(* CODESYS project SMART_HOME_SANDBOX_V2.xml

Project tree, tasks and I/O mapping:
  PLC_A : PLC210, Production association OWEN, order no. 1, version 3.5.17.35
    application Application
      libraries: SysMem, 3.5.17.0 (System); Net Base Services, 3.5.17.0 (3S - Smart Software Solutions GmbH); OwenCommunication, 3.5.11.7 (Production association OWEN); Standard, * (System); AC_ModuleBase, * (3S - Smart Software Solutions GmbH); AC_DataLog, * (3S - Smart Software Solutions GmbH); VisuElem3DPath, 4.1.0.0 (System); VisuElemMeter, 4.1.0.0 (System); VisuElemTrace, 4.1.0.0 (System); VisuElemBase, 4.1.0.0 (System); VisuElems, 4.1.0.0 (System); VisuElemsSpecialControls, 4.1.0.0 (System); VisuElemsWinControls, 4.1.0.0 (System); VisuElemTextEditor, 4.1.0.0 (System); VisuNativeControl, 4.1.0.0 (System); VisuElemsAlarm, 4.1.0.0 (System); VisuElemCamDisplayer, 4.1.0.0 (System); VisuElemsDateTime, 4.1.0.0 (System); VisuElemXYChart, 4.1.0.0 (System); VisuInputs, 4.1.0.0 (System); CmpTargetVisu, 3.5.17.0 (System); Mx210 Assistant, 3.5.11.11 (Production association OWEN)
      task MainTask (cyclic, interval t#20ms, priority 1) calls PRG_PLC_A, PRG_PLC_B, PRG_Main
      task OwenCloudTask (cyclic, interval T#25ms, priority 31) calls OwenStorage.CLOUD_PRG
      task VISU_TASK (cyclic, interval 100 ms, priority 31) calls VisuElems.Visu_Prg
      program PRG_PLC_A [ST]
      program PRG_PLC_B [ST]
    Ethernet : Ethernet, 3S - Smart Software Solutions GmbH, version 3.5.17.0
        settings: IPAddress = [192,168,10,10]; SubnetMask = [255,255,255,0]; GatewayAddress = [192,168,10,1]; MACAddress = [16#00,16#00,16#00,16#00,16#00,16#00]; NetworkInterfaceName = 'ELECTRICAL_ROOM_1F'; NetworkInterfaceName = "ELECTRICAL_ROOM_1F"; SaveCommunicationSettings = TRUE
      Modbus_TCP_Master : Modbus TCP Master, 3S - Smart Software Solutions GmbH, version 3.5.17.0
        MV210_101 : MV210-101, Production association OWEN, version 3.5.11.13
            settings: Unit-ID = 2; IPAddress = [192, 168, 10, 2]
            input  Application.GVL_IO.AI_Temp_Outdoor : InputValue  // Вход 1
            input  Application.GVL_IO.AI_Temp_Outdoor : REAL  // Вход 1.Значение
            input  Application.GVL_IO.AI_Manifold_Temps_Supply[1] : InputValue  // Вход 2
            input  Application.GVL_IO.AI_Manifold_Temps_Supply[1] : REAL  // Вход 2.Значение
            input  Application.GVL_IO.AI_Manifold_Temps_Supply[2] : InputValue  // Вход 3
            input  Application.GVL_IO.AI_Manifold_Temps_Supply[2] : REAL  // Вход 3.Значение
            input  Application.GVL_IO.AI_Manifold_Temps_Supply[3] : InputValue  // Вход 4
            input  Application.GVL_IO.AI_Manifold_Temps_Supply[3] : REAL  // Вход 4.Значение
            input  Application.GVL_IO.AI_Manifold_Temps_Supply[4] : InputValue  // Вход 5
            input  Application.GVL_IO.AI_Manifold_Temps_Supply[4] : REAL  // Вход 5.Значение
            input  Application.GVL_IO.AI_Manifold_Temps_Supply[5] : InputValue  // Вход 6
            input  Application.GVL_IO.AI_Manifold_Temps_Supply[5] : REAL  // Вход 6.Значение
            input  Application.GVL_IO.AI_Methane_LEL[1] : InputValue  // Вход 7
            input  Application.GVL_IO.AI_Methane_LEL[1] : REAL  // Вход 7.Значение
            input  Application.GVL_IO.AI_Methane_LEL[2] : InputValue  // Вход 8
            input  Application.GVL_IO.AI_Methane_LEL[2] : REAL  // Вход 8.Значение
            unmapped channels: Tmp, Исключить модуль из опроса, Флаг ошибки, Записать настройки, Прочитать настройки, Вход 1 (чтение), Вход 2 (чтение), Вход 3 (чтение), Вход 4 (чтение), Вход 5 (чтение), Вход 6 (чтение), Вход 7 (чтение), Вход 8 (чтение), Вход 1 (запись), Вход 2 (запись), Вход 3 (запись), Вход 4 (запись), Вход 5 (запись), Вход 6 (запись), Вход 7 (запись), Вход 8 (запись)
        MK210_301 : MK210-301, Production association OWEN, version 3.5.11.13
            settings: Unit-ID = 3; IPAddress = [192, 168, 10, 3]
            input  Application.GVL_IO.DI_Security_Open[1] : BOOL  // Битовая маска входов.Вход 1
            input  Application.GVL_IO.DI_Security_Open[2] : BOOL  // Битовая маска входов.Вход 2
            input  Application.GVL_IO.DI_Security_Open[3] : BOOL  // Битовая маска входов.Вход 3
            input  Application.GVL_IO.DI_Security_Open[4] : BOOL  // Битовая маска входов.Вход 4
            input  Application.GVL_IO.DI_Security_Open[5] : BOOL  // Битовая маска входов.Вход 5
            input  Application.GVL_IO.DI_Security_Open[6] : BOOL  // Битовая маска входов.Вход 6
            input  Application.GVL_IO.DO_Manifold_Pumps[1] : BOOL  // Битовая маска выходов (чтение).Выход 1
            input  Application.GVL_IO.DO_Manifold_Pumps[2] : BOOL  // Битовая маска выходов (чтение).Выход 2
            input  Application.GVL_IO.DO_Manifold_Pumps[3] : BOOL  // Битовая маска выходов (чтение).Выход 3
            input  Application.GVL_IO.DO_Manifold_Pumps[4] : BOOL  // Битовая маска выходов (чтение).Выход 4
            input  Application.GVL_IO.DO_Manifold_Pumps[5] : BOOL  // Битовая маска выходов (чтение).Выход 5
            input  Application.GVL_IO.DO_Boiler_Enable[1] : BOOL  // Битовая маска выходов (чтение).Выход 6
            input  Application.GVL_IO.DO_Boiler_Enable[2] : BOOL  // Битовая маска выходов (чтение).Выход 7
            output Application.GVL_IO.DO_Manifold_Pumps[1] : BOOL  // Битовая маска выходов (запись).Выход 1
            output Application.GVL_IO.DO_Manifold_Pumps[2] : BOOL  // Битовая маска выходов (запись).Выход 2
            output Application.GVL_IO.DO_Manifold_Pumps[3] : BOOL  // Битовая маска выходов (запись).Выход 3
            output Application.GVL_IO.DO_Manifold_Pumps[4] : BOOL  // Битовая маска выходов (запись).Выход 4
            output Application.GVL_IO.DO_Manifold_Pumps[5] : BOOL  // Битовая маска выходов (запись).Выход 5
            output Application.GVL_IO.DO_Boiler_Enable[1] : BOOL  // Битовая маска выходов (запись).Выход 6
            output Application.GVL_IO.DO_Boiler_Enable[2] : BOOL  // Битовая маска выходов (запись).Выход 7
            output Application.GVL_IO.DO_DHW_Heating_Pump : BOOL  // Битовая маска выходов (запись).Выход 8
            output Application.GVL_IO.AO_Supply_Fans[1] : localTypes:PwmOutputValue  // Коэффициент заполнения ШИМ (запись)
            output Application.GVL_IO.AO_Supply_Fans[2] : localTypes:PwmOutputValue  // Коэффициент заполнения ШИМ (запись)
            output Application.GVL_IO.AO_Supply_Fans[3] : localTypes:PwmOutputValue  // Коэффициент заполнения ШИМ (запись)
            output Application.GVL_IO.AO_Exhaust_Fans[1] : localTypes:PwmOutputValue  // Коэффициент заполнения ШИМ (запись)
            output Application.GVL_IO.AO_Exhaust_Fans[2] : localTypes:PwmOutputValue  // Коэффициент заполнения ШИМ (запись)
            output Application.GVL_IO.AO_Exhaust_Fans[3] : localTypes:PwmOutputValue  // Коэффициент заполнения ШИМ (запись)
            output Application.GVL_IO.AO_Exhaust_Fans[4] : localTypes:PwmOutputValue  // Коэффициент заполнения ШИМ (запись)
            output Application.GVL_IO.AO_Exhaust_Fans[5] : localTypes:PwmOutputValue  // Коэффициент заполнения ШИМ (запись)
            unmapped channels: Tmp, Исключить модуль из опроса, Флаг ошибки, Битовая маска входов, Битовая маска выходов (чтение), Битовая маска выходов (запись), Значение счетчика, Значение счетчика, Значение счетчика, Значение счетчика, Значение счетчика, Значение счетчика, Сбросить счетчик, Сбросить счетчик, Сбросить счетчик, Сбросить счетчик, Сбросить счетчик, Сбросить счетчик, Период ШИМ (чтение), Период ШИМ (чтение), Период ШИМ (чтение), Период ШИМ (чтение), Период ШИМ (чтение), Период ШИМ (чтение), Период ШИМ (чтение), Период ШИМ (чтение), Период ШИМ (запись), Период ШИМ (запись), Период ШИМ (запись), Период ШИМ (запись), Период ШИМ (запись), Период ШИМ (запись), Период ШИМ (запись), Период ШИМ (запись), Коэффициент заполнения ШИМ (чтение), Коэффициент заполнения ШИМ (чтение), Коэффициент заполнения ШИМ (чтение), Коэффициент заполнения ШИМ (чтение), Коэффициент заполнения ШИМ (чтение), Коэффициент заполнения ШИМ (чтение),
              Коэффициент заполнения ШИМ (чтение), Коэффициент заполнения ШИМ (чтение)
        MV210_202 : MV210-202, Production association OWEN, version 3.5.11.13
            settings: Unit-ID = 4; IPAddress = [192, 168, 10, 4]
            input  Application.GVL_IO.DI_Flood_Sensors[1] : BOOL  // Битовая маска входов.Вход 1
            input  Application.GVL_IO.DI_Flood_Sensors[2] : BOOL  // Битовая маска входов.Вход 2
            input  Application.GVL_IO.DI_Flood_Sensors[3] : BOOL  // Битовая маска входов.Вход 3
            input  Application.GVL_IO.DI_Flood_Sensors[4] : BOOL  // Битовая маска входов.Вход 4
            input  Application.GVL_IO.DI_Flood_Sensors[5] : BOOL  // Битовая маска входов.Вход 5
            input  Application.GVL_IO.DI_Flood_Sensors[6] : BOOL  // Битовая маска входов.Вход 6
            input  Application.GVL_IO.DI_Flood_Sensors[7] : BOOL  // Битовая маска входов.Вход 7
            input  Application.GVL_IO.DI_Flood_Sensors[8] : BOOL  // Битовая маска входов.Вход 8
            input  Application.GVL_IO.DI_Flood_Sensors[9] : BOOL  // Битовая маска входов.Вход 9
            input  Application.GVL_IO.DI_Flood_Sensors[10] : BOOL  // Битовая маска входов.Вход 10
            input  Application.GVL_IO.DI_Flood_Sensors[11] : BOOL  // Битовая маска входов.Вход 11
            input  Application.GVL_IO.DI_Flood_Sensors[12] : BOOL  // Битовая маска входов.Вход 12
            input  Application.GVL_IO.DI_Security_Glass[1] : BOOL  // Битовая маска входов.Вход 13
            input  Application.GVL_IO.DI_Security_Glass[2] : BOOL  // Битовая маска входов.Вход 14
            input  Application.GVL_IO.DI_Security_Glass[3] : BOOL  // Битовая маска входов.Вход 15
            input  Application.GVL_IO.DI_Security_Glass[4] : BOOL  // Битовая маска входов.Вход 16
            input  Application.GVL_IO.DI_Security_Glass[5] : BOOL  // Битовая маска входов.Вход 17
            input  Application.GVL_IO.DI_Security_Glass[6] : BOOL  // Битовая маска входов.Вход 18
            input  Application.GVL_IO.DI_Security_Glass[7] : BOOL  // Битовая маска входов.Вход 19
            input  Application.GVL_IO.DI_Security_Glass[8] : BOOL  // Битовая маска входов.Вход 20
            unmapped channels: Tmp, Исключить модуль из опроса, Флаг ошибки, Битовая маска входов, Значение, Значение, Значение, Значение, Значение, Значение, Значение, Значение, Значение счетчика, Значение счетчика, Значение счетчика, Значение счетчика, Значение счетчика, Значение счетчика, Значение счетчика, Значение счетчика, Значение счетчика, Значение счетчика, Значение счетчика, Значение счетчика, Сбросить значение, Сбросить значение, Сбросить значение, Сбросить значение, Сбросить значение, Сбросить значение, Сбросить значение, Сбросить значение, Сбросить счетчик, Сбросить счетчик, Сбросить счетчик, Сбросить счетчик, Сбросить счетчик, Сбросить счетчик, Сбросить счетчик, Сбросить счетчик,
              Сбросить счетчик, Сбросить счетчик, Сбросить счетчик, Сбросить счетчик
        MU210_401 : MU210-401, Production association OWEN, version 3.5.11.13
            settings: Unit-ID = 5; IPAddress = [192, 168, 10, 5]
            output Application.GVL_IO.AO_Manifold_Valves[1] : localTypes:CoefficientPWM  // Коэффициент заполнения ШИМ (запись)
            output Application.GVL_IO.AO_Manifold_Valves[2] : localTypes:CoefficientPWM  // Коэффициент заполнения ШИМ (запись)
            output Application.GVL_IO.AO_Manifold_Valves[3] : localTypes:CoefficientPWM  // Коэффициент заполнения ШИМ (запись)
            output Application.GVL_IO.AO_Manifold_Valves[4] : localTypes:CoefficientPWM  // Коэффициент заполнения ШИМ (запись)
            output Application.GVL_IO.AO_Manifold_Valves[5] : localTypes:CoefficientPWM  // Коэффициент заполнения ШИМ (запись)
            output Application.GVL_IO.AO_Boiler_Setpoint[1] : localTypes:CoefficientPWM  // Коэффициент заполнения ШИМ (запись)
            output Application.GVL_IO.AO_Boiler_Setpoint[2] : localTypes:CoefficientPWM  // Коэффициент заполнения ШИМ (запись)
            unmapped channels: Tmp, Исключить модуль из опроса, Флаг ошибки, Битовая маска выходов (чтение), Битовая маска выходов (запись), Период ШИМ (чтение), Период ШИМ (чтение), Период ШИМ (чтение), Период ШИМ (чтение), Период ШИМ (чтение), Период ШИМ (чтение), Период ШИМ (чтение), Период ШИМ (чтение), Период ШИМ (запись), Период ШИМ (запись), Период ШИМ (запись), Период ШИМ (запись), Период ШИМ (запись), Период ШИМ (запись), Период ШИМ (запись), Период ШИМ (запись), Коэффициент заполнения ШИМ (чтение), Коэффициент заполнения ШИМ (чтение), Коэффициент заполнения ШИМ (чтение), Коэффициент заполнения ШИМ (чтение), Коэффициент заполнения ШИМ (чтение), Коэффициент заполнения ШИМ (чтение), Коэффициент заполнения ШИМ (чтение), Коэффициент заполнения ШИМ (чтение), Коэффициент заполнения ШИМ (запись)
    PLC210_11 : PLC210-11, Production association OWEN, version 3.5.17.3004
        unmapped channels: Канал питания 1, Канал питания 2, Сервисная кнопка, Температура CPU, Переключатель Старт\Стоп, Напряжение батареи часов, Статус батареи часов, Статус ионисторов, Hostname, New Hostame, Set Hostname
      LeftSide : LeftSide-11, Production association OWEN, version 3.5.17.3004
          unmapped channels: Битовая маска входов, Cчётчик импульсов, Cчётчик импульсов, Cчётчик импульсов, Cчётчик импульсов, Cчётчик импульсов, Cчётчик импульсов, Cчётчик импульсов, Cчётчик импульсов, Период импульса, Период импульса, Период импульса, Период импульса, Период импульса, Период импульса, Период импульса, Период импульса, Длительность импульса, Длительность импульса, Длительность импульса, Длительность импульса, Длительность импульса, Длительность импульса, Длительность импульса, Длительность импульса, Статус генератора импульсов, Статус генератора импульсов, Статус генератора импульсов, Статус генератора импульсов, Осталось сгенерировать импульсов, Осталось сгенерировать импульсов, Осталось сгенерировать импульсов, Осталось сгенерировать импульсов, Сброс счётчика импульсов, Сброс счётчика импульсов, Сброс счётчика импульсов, Сброс счётчика импульсов, Сброс счётчика импульсов, Сброс счётчика импульсов, Сброс счётчика импульсов,
            Сброс счётчика импульсов, Битовая маска выходов (запись), Запустить генератор, Запустить генератор, Запустить генератор, Запустить генератор, Количество импульсов генератора (запись), Количество импульсов генератора (запись), Количество импульсов генератора (запись), Количество импульсов генератора (запись), Выход 1, Выход 2, Выход 3, Выход 4, Выход 1, Выход 2, Выход 3, Выход 4, Выход 1, Выход 2, Выход 3, Выход 4, Выход 1, Выход 2, Выход 3, Выход 4
      RightSide : RightSide-11, Production association OWEN, version 3.5.17.3002
          unmapped channels: Наличие связи, Счетчик ошибок, Битовая маска диагностики выходов, Битовая маска выходов (запись)
    OwenRTC : OwenRTC, Production association OWEN, version 3.5.17.3002
        unmapped channels: Year, Month, Day, Hour, Minute, Second, Day of Week, Week of Year, Format Date, Format Time, UTC Offset, NTP Enabled, NTP Error, System Timer, Date And Time, Operating Time, New Year, New Month, New Day, New Hour, New Minute, New Second, New UTC Offset, Set Settings DT, Enable NTP, Prefer Server, Sync time by NTP
    OwenCloud : OwenCloud, Production association OWEN, version 3.5.17.3004
        unmapped channels: OwenCloud enabled, Folder error, Symbol error, No Symbol Config, Status, Warning Big Symbol Name, Warning Symbol Name, Symbol Count, Enable OwenCloud
    Buzzer : Buzzer, Production association OWEN, version 3.5.17.3002
        unmapped channels: Buzzer enabled, Enable Buzzer, Sound frequency
    Drives : Drives, Production association OWEN, version 3.5.17.3003
        unmapped channels: FS size, FS used, FS free, USB Mounted, USB Unmount done, USB size, USB used, USB free, MMC Mounted, MMC Unmount done, MMC size, MMC used, MMC free, FS wear, USB FS Info, MMC FS Info, Enable Drives, USB Unmount, MMC Unmount
    Debug : Debug, Production association OWEN, version 3.5.17.3002
        unmapped channels: RAM used, RAM free, Open files, Processor usage, Core temp, Enable Debug, Debug pause
    Info : Info, Production association OWEN, version 3.5.17.3002
        unmapped channels: VENDOR, DEVICE, SERIAL, RUNTIME, FIRMWARE, LINUX, TARGET, PROJECT, AUTHOR, VERSION, PROFILE, LASTCHANGES
    Watchdog : Watchdog, Production association OWEN, version 3.5.17.3002
        unmapped channels: Exception Handling, Last Exception Code, Last Exception Description, Last Exception Time, Hardware Watchdog Flag, Power Reboot Count, Watchdog Reboot Count, Exception Reboot Count, Command Reboot Count, Reboot, Reset Counters
  libraries: VisuSymbols, 4.1.0.0 (System); SysFileAsync, 3.5.17.0 (System); SysFile, 3.5.17.0 (System); Mx210 Assistant, 3.5.11.11 (Production association OWEN); VisuElemsDateTime Interfaces, 4.1.0.0 (Intern)
  DUT/
    ENUM/
      data type E_ALERT_PRIORITY
      data type E_Debug_Log_Level
      data type E_Lifetime_Device_Type
      data type E_Outdoor_Mode
      data type E_PLC_ROLE
      data type E_Rule_Action_Type
      data type E_Rule_Comparison
      data type E_Rule_Condition_Type
      data type E_SCENARIO_TYPE
      data type E_SENSOR_TYPE
      data type E_Trend_Parameter_Type
      data type E_TwoFactor_Method
      data type E_Valve_Test_Result
      data type E_VALVE_TYPE
      data type E_VENTILATION_LOCATION
      data type E_VENTILATION_UNIT_TYPE
      data type E_WEATHER_COMPENSATION_METHOD
      data type E_Zone_Access_Level
    STRUCT/
      data type ST_Astro_Time
      data type ST_BlackBox_Record
      data type ST_Boiler_Status
      data type ST_Component_Maintenance
      data type ST_Debug_Logger_Config
      data type ST_Debug_Log_Record
      data type ST_Device_Health
      data type ST_DHW_Config
      data type ST_DHW_Status
      data type ST_Flood_Config
      data type ST_Flood_Global_Config
      data type ST_FloorHeating_Circuit_Config
      data type ST_FloorHeating_Global_Config
      data type ST_FloorHeating_Manifold_Config
      data type ST_Gas_Valve_Configuration
      data type ST_Gateway_Command
      data type ST_Heating_Config
      data type ST_History_Record
      data type ST_Lifetime_Status
      data type ST_Maintenance_Access_Config
      data type ST_Manifold_Status
      data type ST_Operator_Zone_Rights
      data type ST_Outdoor_Zone_Config
      data type ST_Owen_Analog_Value
      data type ST_Rule_Action
      data type ST_Scenario_Config
      data type ST_Scenario_Transition_Config
      data type ST_Security_Config
      data type ST_Security_Global_Config
      data type ST_Security_Zone_State
      data type ST_Sensor_Calibration_Record
      data type ST_State_Snapshot
      data type ST_System_State_Summary
      data type ST_Tariff_Config
      data type ST_Trend_Config
      data type ST_Trend_Data
      data type ST_Trend_Header
      data type ST_Trend_History_Record
      data type ST_TwoFactor_Auth_State
      data type ST_TwoFactor_Data
      data type ST_User_Rule
      data type ST_Valve_Test_Config
      data type ST_Ventilation_Config
      data type ST_Ventilation_Global_Config
      data type ST_Ventilation_Scenario_Mode
      data type ST_Ventilation_Unit
      data type ST_Ventilation_Unit_Config
      data type ST_Zone_Sensors
  GVL/
    global variables GVL_BlackBox
    global variables GVL_Constants
    global variables GVL_Diagnostics
    global variables GVL_Global_Variables
    global variables GVL_HMI_Config
    global variables GVL_IO
    global variables GVL_Vars
  POUs/
    function block FB_AccessCode_Manager [ST]
    function block FB_Access_Control [ST]
    function block FB_Astro_Timer [ST]
    function block FB_BlackBox_Recorder [ST]
    function block FB_Boiler_Cascade_Controller [ST]
    function block FB_Boiler_Cascade_Manager [ST]
    function block FB_Calibration_Manager [ST]
    function block FB_CO_Detector [ST]
    function block FB_CRC32_Calculator [ST]: Calculate, InitTable
    function block FB_Debug_Logger [ST]
    function block FB_Device_Predictive_Diag [ST]
    function block FB_DHW_Manager [ST]
    function block FB_Emergency_Valve_Open [ST]
    function block FB_Exhaust_Ventilation_Controller [ST]
    function block FB_Flood_Detector [ST]
    function block FB_FloorHeating_Controller [ST]
    function block FB_FloorHeating_Freeze_Protection [ST]
    function block FB_FloorHeating_Overheat_Protection [ST]
    function block FB_Gas_Methane_Detector [ST]
    function block FB_Gas_Smoke_Manager [ST]
    function block FB_Gas_Valve_Controller [ST]: CloseValve, GetStatus, OpenValve
    function block FB_Gateway_Interface [ST]
    function block FB_Heating_System_Manager [ST]
    function block FB_History_Manager [ST]
    function block FB_Lifetime_Predictor [ST]
    function block FB_Lighting_Blinds_Manager [ST]
    function block FB_Maintenance_Access [ST]
    function block FB_Manifold_Mixing_Valve_Controller [ST]
    function block FB_Manifold_Pump_Controller [ST]
    function block FB_Manual_Valve_Control [ST]
    function block FB_NVRAM_Manager [ST]
    function block FB_Outdoor_Lighting_Controller [ST]
    function block FB_PID_Controller [ST]
    function block FB_PLC_Heartbeat [ST]
    function block FB_Presence_Playback [ST]
    function block FB_Presence_Simulator [ST]
    function block FB_Pre_Departure_Heating [ST]
    function block FB_Random_Generator [ST]: Random_Int_Range
    function block FB_Scenario_Manager [ST]
    function block FB_Scenario_Transition_Controller [ST]
    function block FB_Security_Alarm [ST]: CheckPerimeter
    function block FB_Security_System [ST]
    function block FB_Security_System_Manager [ST]
    function block FB_Sensor_Calibration_Processor [ST]
    function block FB_Sensor_Distribution [ST]
    function block FB_Simulation_Manager [ST]
    function block FB_Smoke_Detector [ST]
    function block FB_SMS_Notification [ST]
    function block FB_State_Manager [ST]
    function block FB_State_Snapshot_Manager [ST]
    function block FB_State_Snapshot_NVRAM [ST]
    function block FB_Supply_Ventilation_Controller [ST]
    function block FB_Trend_Analyzer [ST]
    function block FB_TwoFactor_Auth [ST]
    function block FB_User_Rule_Engine [ST]
    function block FB_Valve_Test [ST]
    function block FB_Ventilation_System_Manager [ST]
    function block FB_Water_Leakage_Manager [ST]
    function block FB_Water_Valve_Controller [ST]: CloseValve, GetStatus, OpenValve
    function block FB_Zone_Access_Manager [ST]: CheckAccess
  text list GlobalTextList
  interface IValveController: CloseValve, GetStatus, OpenValve
  program PRG_Main [ST]
  visualisation Visualization
*)

// DUT/ENUM/E_ALERT_PRIORITY
{attribute 'qualified_only'}
{attribute 'strict'}
TYPE E_ALERT_PRIORITY :
(
    ALERT_PRIORITY_NONE := 0,
    ALERT_PRIORITY_LOW := 1,
    ALERT_PRIORITY_MEDIUM := 2,
    ALERT_PRIORITY_HIGH := 3,
    ALERT_PRIORITY_CRITICAL := 4
) BYTE;
END_TYPE

// DUT/ENUM/E_Debug_Log_Level
{attribute 'qualified_only'}
{attribute 'strict'}
TYPE E_Debug_Log_Level :
(
    LOG_LEVEL_MINIMAL := 0,
    LOG_LEVEL_NORMAL := 1,
    LOG_LEVEL_VERBOSE := 2,
    LOG_LEVEL_DEBUG := 3
) BYTE;
END_TYPE

// DUT/ENUM/E_Lifetime_Device_Type
{attribute 'qualified_only'}
{attribute 'strict'}
TYPE E_Lifetime_Device_Type :
(
    LIFETIME_DEVICE_PUMP := 1,
    LIFETIME_DEVICE_FAN  := 2
) BYTE;
END_TYPE

// DUT/ENUM/E_Outdoor_Mode
{attribute 'qualified_only'}
{attribute 'strict'}
TYPE E_Outdoor_Mode :
(
    OUTDOOR_MODE_AUTO := 0,
    OUTDOOR_MODE_PARTY := 1,
    OUTDOOR_MODE_SECURITY := 2,
    OUTDOOR_MODE_ECONOMY := 3,
    OUTDOOR_MODE_MANUAL := 4
) BYTE;
END_TYPE

// DUT/ENUM/E_PLC_ROLE
{attribute 'qualified_only'}
{attribute 'strict'}
TYPE E_PLC_ROLE :
(
    ROLE_UNDEFINED := 0,
    ROLE_ACTIVE := 1,
    ROLE_STANDBY := 2,
    ROLE_OFFLINE := 3
) USINT;
END_TYPE

// DUT/ENUM/E_Rule_Action_Type
{attribute 'qualified_only'}
{attribute 'strict'}
TYPE E_Rule_Action_Type :
(
    ACTION_NONE := 0,
    ACTION_SET_FLOOR_HEATING := 1,
    ACTION_SET_LIGHTING_BASE := 2,
    ACTION_SET_LIGHTING_ACCENT := 3,
    ACTION_SET_SOCKET := 4,
    ACTION_SET_VENTILATION := 5,
    ACTION_SET_BLINDS := 6,
    ACTION_ACTIVATE_SCENARIO := 7,
    ACTION_TOGGLE_LIGHTING := 8,
    ACTION_TOGGLE_SOCKET := 9
) BYTE;
END_TYPE

// DUT/ENUM/E_Rule_Comparison
{attribute 'qualified_only'}
{attribute 'strict'}
TYPE E_Rule_Comparison :
(
    COMP_NONE := 0,
    COMP_EQ := 1,
    COMP_GT := 2,
    COMP_LT := 3,
    COMP_GE := 4,
    COMP_LE := 5,
    COMP_IN_RANGE := 6,
    COMP_TRUE := 7,
    COMP_FALSE := 8
) BYTE;
END_TYPE

// DUT/ENUM/E_Rule_Condition_Type
{attribute 'qualified_only'}
{attribute 'strict'}
TYPE E_Rule_Condition_Type :
(
    COND_NONE := 0,
    COND_AIR_TEMP := 1,
    COND_FLOOR_TEMP := 2,
    COND_HUMIDITY := 3,
    COND_CO2 := 4,
    COND_METHANE := 5,
    COND_CO := 6,
    COND_DOOR_WINDOW := 7,
    COND_FLOOD := 8,
    COND_SMOKE := 9,
    COND_MOTION := 10,
    COND_TIME_OF_DAY := 11,
    COND_DAY_OF_WEEK := 12,
    COND_AND := 13, // Логическое И (Rule Chaining)
    COND_OR := 14   // Логическое ИЛИ (Rule Chaining)
) BYTE;
END_TYPE

// DUT/ENUM/E_SCENARIO_TYPE
{attribute 'qualified_only'}
{attribute 'strict'}
TYPE E_SCENARIO_TYPE :
(
    SCENARIO_NONE := 0,
    SCENARIO_MORNING := 1,
    SCENARIO_EVENING := 2,
    SCENARIO_AWAY := 3,
    SCENARIO_PARTY := 4,
    SCENARIO_SLEEP := 5,
    SCENARIO_EMERGENCY := 6,
    SCENARIO_PRESENCE := 7
) BYTE;
END_TYPE

// DUT/ENUM/E_SENSOR_TYPE
{attribute 'qualified_only'}
{attribute 'strict'}
TYPE E_SENSOR_TYPE :
(
  SENSOR_TYPE_NONE := 0,
  SENSOR_TYPE_DOOR_WINDOW := 5,
  SENSOR_TYPE_GLASS_BREAK := 6,
  SENSOR_TYPE_FLOOD := 7,
  SENSOR_TYPE_SMOKE := 8,
  SENSOR_TYPE_GAS_METHANE := 1,
  SENSOR_TYPE_GAS_CO := 2,
  SENSOR_TYPE_TEMP_FLOOR := 3,
  SENSOR_TYPE_TEMP_AIR := 4
) USINT;
END_TYPE

// DUT/ENUM/E_Trend_Parameter_Type
{attribute 'qualified_only'}
{attribute 'strict'}
TYPE E_Trend_Parameter_Type :
(
    TREND_PARAM_NONE := 0,
    TREND_PARAM_TEMP_AIR := 1,
    TREND_PARAM_TEMP_FLOOR := 2,
    TREND_PARAM_PRESSURE := 3,
    TREND_PARAM_PUMP_CURRENT := 4,
    TREND_PARAM_GAS_METHANE := 5,
    TREND_PARAM_GAS_CO := 6
) BYTE;
END_TYPE

// DUT/ENUM/E_TwoFactor_Method
{attribute 'qualified_only'}
{attribute 'strict'}
TYPE E_TwoFactor_Method :
(
    TF_METHOD_NONE := 0,
    TF_METHOD_RFID := 1,
    TF_METHOD_TOTP := 2,
    TF_METHOD_BOTH := 3
) BYTE;
END_TYPE

// DUT/ENUM/E_Valve_Test_Result
{attribute 'qualified_only'}
{attribute 'strict'}
TYPE E_Valve_Test_Result :
(
    TEST_RESULT_NONE := 0,
    TEST_RESULT_PASSED := 1,
    TEST_RESULT_CURRENT_DEVIATION := 2,
    TEST_RESULT_TIME_DEVIATION := 3,
    TEST_RESULT_STALL := 4,
    TEST_RESULT_LIMIT_SWITCH_FAIL := 5,
    TEST_RESULT_ABORTED := 6
) BYTE;
END_TYPE

// DUT/ENUM/E_VALVE_TYPE
{attribute 'qualified_only'}
{attribute 'strict'}
TYPE E_VALVE_TYPE :
(
  VALVE_NC := 1,  // Нормально-закрытый
  VALVE_NO := 2   // Нормально-открытый
) USINT;
END_TYPE

// DUT/ENUM/E_VENTILATION_LOCATION
{attribute 'qualified_only'}
{attribute 'strict'}
TYPE E_VENTILATION_LOCATION :
(
  VENT_LOCATION_NONE := 0,
  VENT_LOCATION_BASEMENT_GAME_ROOM := 1,
  VENT_LOCATION_BASEMENT_GYM := 2,
  VENT_LOCATION_BASEMENT_BOILER_ROOM := 3,
  VENT_LOCATION_BATHROOM_1F := 4,
  VENT_LOCATION_BATHROOM_2F := 5,
  VENT_LOCATION_MASTER_BATHROOM := 6,
  VENT_LOCATION_LAUNDRY := 7,
  VENT_LOCATION_KITCHEN := 8
) BYTE;
END_TYPE

// DUT/ENUM/E_VENTILATION_UNIT_TYPE
{attribute 'qualified_only'}
{attribute 'strict'}
TYPE E_VENTILATION_UNIT_TYPE :
(
  VENTILATION_TYPE_NONE := 0,
  VENTILATION_TYPE_SUPPLY := 1,
  VENTILATION_TYPE_EXHAUST := 2
) USINT;
END_TYPE

// DUT/ENUM/E_WEATHER_COMPENSATION_METHOD
{attribute 'qualified_only'}
{attribute 'strict'}
TYPE E_WEATHER_COMPENSATION_METHOD :
(
  WEATHER_COMP_NONE := 0,
  WEATHER_COMP_OUTDOOR_RESET := 1
) USINT;
END_TYPE

// DUT/ENUM/E_Zone_Access_Level
{attribute 'qualified_only'}
{attribute 'strict'}
TYPE E_Zone_Access_Level :
(
    ZONE_ACCESS_NONE := 0,
    ZONE_ACCESS_VIEW := 1,
    ZONE_ACCESS_CONTROL := 2,
    ZONE_ACCESS_CONFIG := 3,
    ZONE_ACCESS_FULL := 4
) BYTE;
END_TYPE

// DUT/STRUCT/ST_Astro_Time
TYPE ST_Astro_Time :
STRUCT
    sunrise_ms : UDINT := 0;
    sunset_ms : UDINT := 0;
    is_daylight : BOOL := FALSE;
END_STRUCT
END_TYPE

// DUT/STRUCT/ST_BlackBox_Record
TYPE ST_BlackBox_Record :
STRUCT
    Timestamp : UDINT;
    Gas_Methane_LEL : REAL;
    Gas_CO_PPM : REAL;
    Flood_Active : BOOL;
    Fire_Active : BOOL;
    Valve_Gas_Status : BYTE;
    Valve_Water_Status : BYTE;
    PLC_Active_ID : BYTE;
END_STRUCT
END_TYPE

// DUT/STRUCT/ST_Boiler_Status
TYPE ST_Boiler_Status :
STRUCT
    Active : BOOL;
    Running : BOOL;
    Error : BOOL;
    Power_Percent : REAL;
    Current_Power : REAL;
    Work_Seconds : UDINT;
    Work_Hours : REAL;
    Resource_Percent : REAL := 100.0;
    Last_Start : DT;
END_STRUCT
END_TYPE

// DUT/STRUCT/ST_Component_Maintenance
TYPE ST_Component_Maintenance :
STRUCT
    Is_Faulty : BOOL;        // Устройство неисправно
    Is_In_Maintenance : BOOL; // Выведено в ремонт вручную
    Fallback_Value : REAL;   // Значение для подстановки (0-100% или температура)
    Use_Last_Good_Value : BOOL; // Использовать последнее достоверное значение
END_STRUCT
END_TYPE

// DUT/STRUCT/ST_Debug_Logger_Config
TYPE ST_Debug_Logger_Config :
STRUCT
    enabled : BOOL;
    sampling_period_ms : UDINT := 1000;
END_STRUCT
END_TYPE

// DUT/STRUCT/ST_Debug_Log_Record
TYPE ST_Debug_Log_Record :
STRUCT
    timestamp_ms : UDINT;
    level : BYTE; // E_Debug_Log_Level
    source_id : BYTE;
    event_code : WORD;
    value_int : UDINT;
    value_real : REAL;
    text : STRING(80);
    crc32 : DWORD;
END_STRUCT
END_TYPE

// DUT/STRUCT/ST_Device_Health
TYPE ST_Device_Health :
STRUCT
    Health_Score : BYTE := 100; // 0..100%
    Total_Runtime_Hours : UDINT;
    Starts_Count : UDINT;
    Last_Start_Current : REAL;
    Avg_Start_Current : REAL;
    Maintenance_Required : BOOL;
    Warning_Message : STRING(50);
END_STRUCT
END_TYPE

// DUT/STRUCT/ST_DHW_Config
TYPE ST_DHW_Config :
STRUCT
    Target_Temp : REAL := 55.0;
    Hysteresis : REAL := 2.0;
    Circulation_Schedule_Enabled : BOOL := TRUE;
    Circulation_Start : TOD := TOD#06:00;
    Circulation_End : TOD := TOD#23:00;
    Anti_Legionella_Enabled : BOOL := TRUE;
    Anti_Legionella_Day : UINT := 7; // Воскресенье
END_STRUCT
END_TYPE

// DUT/STRUCT/ST_DHW_Status
TYPE ST_DHW_Status :
STRUCT
    Temp : REAL;
    Pressure : REAL;
    Heating_Pump_On : BOOL;
    Circ_Pump_On : BOOL;
    Error : BOOL;
    Error_ID : WORD;
END_STRUCT
END_TYPE

// DUT/STRUCT/ST_Flood_Config
TYPE ST_Flood_Config :
STRUCT
    Emergency_Two_Stage_Enabled : BOOL := TRUE; // ТЗ 4.4
    Valve_Test_Period_Days : UINT := 7; // ТЗ 12.2
    Current_Threshold_MA : REAL := 500.0; // Порог тока для диагностики
END_STRUCT
END_TYPE

// DUT/STRUCT/ST_Flood_Global_Config
TYPE ST_Flood_Global_Config :
STRUCT
    valve_types : ARRAY[1..3] OF E_VALVE_TYPE := [3(E_VALVE_TYPE.VALVE_NC)];
    min_duration_ms : UDINT := 30000;
END_STRUCT
END_TYPE

// DUT/STRUCT/ST_FloorHeating_Circuit_Config
TYPE ST_FloorHeating_Circuit_Config :
STRUCT
    circuit_id : BYTE := 0;
    zone : BYTE := 0;
    design_temp : REAL := 35.0;
    min_temp : REAL := 20.0;
    max_temp : REAL := 45.0;
    pid_kp : REAL := 2.0;
END_STRUCT
END_TYPE

// DUT/STRUCT/ST_FloorHeating_Global_Config
TYPE ST_FloorHeating_Global_Config :
STRUCT
    enable_floor_heating : BOOL := TRUE;
    anti_freeze_temp : REAL := 7.0;
    overheat_temp : REAL := 45.0;
    weather_compensation_enabled : BOOL := TRUE;
    total_circuits : BYTE := 16;
END_STRUCT
END_TYPE

// DUT/STRUCT/ST_FloorHeating_Manifold_Config
TYPE ST_FloorHeating_Manifold_Config :
STRUCT
    manifold_id : BYTE;
    location : STRING(30);
    nominal_flow : REAL;
    enable_pump : BOOL;
    circuits : ARRAY[1..4] OF ST_FloorHeating_Circuit_Config;
END_STRUCT
END_TYPE

// DUT/STRUCT/ST_Gas_Valve_Configuration
TYPE ST_Gas_Valve_Configuration :
STRUCT
    valve_id : BYTE := 0;
    valve_type : E_VALVE_TYPE := E_VALVE_TYPE.VALVE_NC;
    close_time_seconds : UDINT := 10;
    open_time_seconds : UDINT := 10;
    emergency_open_allowed : BOOL := FALSE;
END_STRUCT
END_TYPE

// DUT/STRUCT/ST_Gateway_Command
TYPE ST_Gateway_Command :
STRUCT
    command_id : UDINT;
    timestamp_ms : UDINT;
    operator_id : STRING(10);
    command_type : BYTE;
    target_zone : BYTE;
    target_value : REAL;
    target_on_off : BOOL;
    target_scenario : E_SCENARIO_TYPE;
    target_armed : BOOL;
    crc32 : DWORD;
END_STRUCT
END_TYPE

// DUT/STRUCT/ST_Heating_Config
TYPE ST_Heating_Config :
STRUCT
    Weather_Comp_Enabled : BOOL := TRUE;
    Weather_Coef : REAL := 0.1;
    Freeze_Threshold : REAL := 7.0;
    Overheat_Threshold : REAL := 45.0;
    Night_Reduction : REAL := 3.0;
    Target_Floor_Temp : REAL := 28.0;
    Target_Room_Temp : REAL := 22.0;
    Hysteresis : REAL := 0.5;
END_STRUCT
END_TYPE

// DUT/STRUCT/ST_History_Record
TYPE ST_History_Record :
STRUCT
    timestamp_ms : UDINT := 0;
    event_code : WORD := 0;
    event_value : REAL := 0.0;
    unit : BYTE := 0;
    zone_id : BYTE := 0;
    operator_id : STRING(10) := '';
    priority : E_ALERT_PRIORITY := E_ALERT_PRIORITY.ALERT_PRIORITY_NONE;
END_STRUCT
END_TYPE

// DUT/STRUCT/ST_Lifetime_Status
TYPE ST_Lifetime_Status :
STRUCT
    device_id : BYTE;
    runtime_hours : UDINT;
    start_count : UDINT;
    remaining_hours : UDINT;
    remaining_percent : BYTE;
    maintenance_required : BOOL;
    last_calc_timestamp : UDINT;
END_STRUCT
END_TYPE

// DUT/STRUCT/ST_Maintenance_Access_Config
TYPE ST_Maintenance_Access_Config :
STRUCT
    maintenance_enabled : BOOL := FALSE;
    max_duration_minutes : UDINT := 60;
    requires_two_person : BOOL := TRUE;
    access_level_required : BYTE := 2;
END_STRUCT
END_TYPE

// DUT/STRUCT/ST_Manifold_Status
TYPE ST_Manifold_Status :
STRUCT
    Pump_On : BOOL;
    Pump_Current : REAL;
    Pressure : REAL;
    Temp_Supply : REAL;
    Temp_Return : REAL;
    Valve_Pos : REAL; // 0-100%
    Error : BOOL;
    Error_ID : WORD;
END_STRUCT
END_TYPE

// DUT/STRUCT/ST_Operator_Zone_Rights
TYPE ST_Operator_Zone_Rights :
STRUCT
    operator_id : STRING(10);
    global_access_level : BYTE := 0;
    zone_masks : ARRAY[1..18] OF DWORD;
    last_modified : UDINT;
END_STRUCT
END_TYPE

// DUT/STRUCT/ST_Outdoor_Zone_Config
TYPE ST_Outdoor_Zone_Config :
STRUCT
    zone_id : BYTE := 0;
    lighting_circuit_id : BYTE := 0;
    auto_enabled : BOOL := TRUE;
    party_mode_enabled : BOOL := FALSE;
END_STRUCT
END_TYPE

// DUT/STRUCT/ST_Owen_Analog_Value
TYPE ST_Owen_Analog_Value :
STRUCT
    rValue : REAL;         // Измеренное значение
    uiCycleTime : UINT;    // Циклическое время
    wStatus : WORD;        // Код статуса (ANALOG_SENSOR_ERRORS)
END_STRUCT
END_TYPE

// DUT/STRUCT/ST_Rule_Action
TYPE ST_Rule_Action :
STRUCT
    Active : BOOL;
    Target_ID : BYTE;
    Value : REAL;
END_STRUCT
END_TYPE

// DUT/STRUCT/ST_Scenario_Config
TYPE ST_Scenario_Config :
STRUCT
    scenario_id : E_SCENARIO_TYPE;
    lighting_level_base : BYTE := 100;
    lighting_level_accent : BYTE := 100;
    floor_heating_adjust_celsius : REAL := 0.0;
    ventilation_speed_percent : BYTE := 50;
    sockets_enabled : BOOL := TRUE;
    blinds_position_percent : BYTE := 0;
END_STRUCT
END_TYPE

// DUT/STRUCT/ST_Scenario_Transition_Config
TYPE ST_Scenario_Transition_Config :
STRUCT
    current_scenario : E_SCENARIO_TYPE;
    target_scenario : E_SCENARIO_TYPE;
    min_duration_minutes : UDINT := 5;
    transition_allowed : BOOL := FALSE;
END_STRUCT
END_TYPE

// DUT/STRUCT/ST_Security_Config
TYPE ST_Security_Config :
STRUCT
    PIN_Code : STRING(4) := '1234';
    Max_Attempts : UINT := 3;
    Entry_Delay_S : UINT := 45;
    Two_Factor_Enabled : BOOL := FALSE;
    Two_Stage_Mode : BOOL := TRUE; // ТЗ 3.4
    Confirmation_Timeout_S : UINT := 120; // ТЗ 3.4 (60-300с)
    Phones : ARRAY[1..5] OF STRING(15);
    
    // Управление доступом
    gate_open_pulse_ms : UDINT := 1000;
    wicket_open_pulse_ms : UDINT := 1000;
    lock_open_pulse_ms : UDINT := 1000;
    lock_close_pulse_ms : UDINT := 1000;
END_STRUCT
END_TYPE

// DUT/STRUCT/ST_Security_Global_Config
TYPE ST_Security_Global_Config :
STRUCT
    entry_delay_seconds : UDINT := 30;
    exit_delay_seconds : UDINT := 60;
    alarm_duration_seconds : UDINT := 180;
    two_person_timeout_seconds : UDINT := 120;
    max_access_attempts : BYTE := 3;
    auto_arm_enabled : BOOL := FALSE;
    auto_arm_time_ms : UDINT := 0;
    
    // ТЗ: Управление доступом
    gate_open_pulse_ms : UDINT := 1000;
    wicket_open_pulse_ms : UDINT := 1000;
    lock_open_pulse_ms : UDINT := 1000;
    lock_close_pulse_ms : UDINT := 1000;
END_STRUCT
END_TYPE

// DUT/STRUCT/ST_Security_Zone_State
TYPE ST_Security_Zone_State :
STRUCT
    Armed : BOOL;
    Alarm : BOOL;
    Bypassed : BOOL;
    Last_Trigger_Time : DT;
    Trigger_Count : UINT;
END_STRUCT
END_TYPE

// DUT/STRUCT/ST_Sensor_Calibration_Record
TYPE ST_Sensor_Calibration_Record :
STRUCT
    sensor_id : UDINT := 0;
    sensor_type : E_SENSOR_TYPE;
    zone_id : BYTE := 0;
    offset : REAL := 0.0;
    multiplier : REAL := 1.0;
    last_calibration_timestamp : UDINT := 0;
    verification_passed : BOOL := FALSE;
END_STRUCT
END_TYPE

// DUT/STRUCT/ST_State_Snapshot
TYPE ST_State_Snapshot :
STRUCT
    timestamp_ms : UDINT := 0;
    operator_id : STRING(10) := '';
    scenario_id : E_SCENARIO_TYPE := E_SCENARIO_TYPE.SCENARIO_NONE;
    lighting_levels : ARRAY[1..16] OF BYTE;
    floor_heating_setpoints : ARRAY[1..16] OF REAL;
    alarm_active : BOOL := FALSE;
    crc32 : DWORD := 0;
END_STRUCT
END_TYPE

// DUT/STRUCT/ST_System_State_Summary
TYPE ST_System_State_Summary :
STRUCT
    Outdoor_Temp : REAL;
    Indoor_Temp : ARRAY[1..16] OF REAL;
    Floor_Temps : ARRAY[1..16] OF REAL;
    Humidity : ARRAY[1..8] OF REAL;
    CO2 : ARRAY[1..8] OF REAL;
    Gas_Alarm : BOOL;
    Flood_Alarm : BOOL;
    Fire_Alarm : BOOL;
    Security_Armed : BOOL;
END_STRUCT
END_TYPE

// DUT/STRUCT/ST_Tariff_Config
TYPE ST_Tariff_Config :
STRUCT
    Enabled : BOOL := FALSE;
    Night_Start_Hour : UINT := 23; // 23:00
    Night_End_Hour : UINT := 7;    // 07:00
    Boost_Delta : REAL := 2.0;     // На сколько градусов поднять уставку ночью
END_STRUCT
END_TYPE

// DUT/STRUCT/ST_Trend_Config
TYPE ST_Trend_Config :
STRUCT
    param_type : BYTE; // E_Trend_Parameter_Type
    zone_id : BYTE;
    enabled : BOOL;
    deviation_threshold_percent : REAL := 10.0;
    history_days : UDINT := 7;
END_STRUCT
END_TYPE

// DUT/STRUCT/ST_Trend_Data
TYPE ST_Trend_Data :
STRUCT
    config : ST_Trend_Config;
    record_count : UDINT;
    write_index : UDINT;
    sum_values : REAL;
    crc32 : DWORD;
END_STRUCT
END_TYPE

// DUT/STRUCT/ST_Trend_Header
TYPE ST_Trend_Header :
STRUCT
    parameter_type : BYTE; // E_Trend_Parameter_Type
    zone_id : BYTE := 0;
    records_count : UDINT := 0;
    average_value : REAL := 0.0;
    min_value : REAL := 0.0;
    max_value : REAL := 0.0;
END_STRUCT
END_TYPE

// DUT/STRUCT/ST_Trend_History_Record
TYPE ST_Trend_History_Record :
STRUCT
    timestamp_ms : UDINT := 0;
    value : REAL := 0.0;
END_STRUCT
END_TYPE

// DUT/STRUCT/ST_TwoFactor_Auth_State
TYPE ST_TwoFactor_Auth_State :
STRUCT
    operator_id : STRING(10);
    is_pending : BOOL; // Ожидание ввода 2-го фактора
    start_time : UDINT;
    timeout_ms : UDINT := 60000;
END_STRUCT
END_TYPE

// DUT/STRUCT/ST_TwoFactor_Data
TYPE ST_TwoFactor_Data :
STRUCT
    operator_id : STRING(10);
    AuthMethod : BYTE; // E_TwoFactor_Method
    rfid_tag : STRING(20);
    totp_secret : STRING(32);
    last_modified : UDINT;
END_STRUCT
END_TYPE

// DUT/STRUCT/ST_User_Rule
TYPE ST_User_Rule :
STRUCT
    Enabled : BOOL;
    Condition_Type : BYTE; // 1-Temp, 2-Hum, 3-CO2, 4-Security, 5-Time
    Condition_Op : BYTE;   // 1:>, 2:<, 3:=
    Condition_Value : REAL;
    Action_Target_ID : BYTE;
    Action_Value : REAL;
    Action_Type : BYTE;    // 1-SetTemp, 2-Switch, 3-Scenario
    Priority : BYTE;       // ТЗ 7.4: Приоритет (0-255)
END_STRUCT
END_TYPE

// DUT/STRUCT/ST_Valve_Test_Config
TYPE ST_Valve_Test_Config :
STRUCT
    valve_id : BYTE := 0;
    test_interval_days : UDINT := 7;
    nominal_current_a : REAL := 0.5;
    Nominal_Current : REAL := 0.5;
    nominal_close_time_sec : REAL := 10.0;
    enabled : BOOL := TRUE;
END_STRUCT
END_TYPE

// DUT/STRUCT/ST_Ventilation_Config
TYPE ST_Ventilation_Config :
STRUCT
    CO2_Threshold : REAL := 800.0;
    Humidity_Threshold : REAL := 65.0;
    Night_Mode_Start : TOD := TOD#23:00;
    Night_Mode_End : TOD := TOD#07:00;
END_STRUCT
END_TYPE

// DUT/STRUCT/ST_Ventilation_Global_Config
TYPE ST_Ventilation_Global_Config :
STRUCT
    enable_ventilation : BOOL := TRUE;
    total_units : BYTE := 8;
    default_supply_speed : BYTE := 40;
    default_exhaust_speed : BYTE := 40;
END_STRUCT
END_TYPE

// DUT/STRUCT/ST_Ventilation_Scenario_Mode
TYPE ST_Ventilation_Scenario_Mode :
STRUCT
  Scenario_ID : BYTE;
  Scenario_Priority : BYTE;
  Fire_Alarm : BOOL;
  Methane_Alarm : BOOL;
  Smoke_Detected : BOOL;
  Exhaust_Modes : ARRAY[1..5] OF BYTE;
  Supply_Modes : ARRAY[1..3] OF BYTE;
END_STRUCT
END_TYPE

// DUT/STRUCT/ST_Ventilation_Unit
TYPE ST_Ventilation_Unit :
STRUCT
    Enabled : BOOL;
    Speed_Percent : REAL;
    Filter_Dirty : BOOL;
    Error : BOOL;
    Mode : BYTE; // 0-Eco, 1-Std, 2-Int, 3-Emergency
END_STRUCT
END_TYPE

// DUT/STRUCT/ST_Ventilation_Unit_Config
TYPE ST_Ventilation_Unit_Config :
STRUCT
    unit_id : BYTE := 0;
    unit_type : E_VENTILATION_UNIT_TYPE;
    location : E_VENTILATION_LOCATION;
    min_speed : BYTE := 20;
    max_speed : BYTE := 100;
    Threshold_Hum : REAL := 65.0;
    has_smoke_detector : BOOL := FALSE;
END_STRUCT
END_TYPE

// DUT/STRUCT/ST_Zone_Sensors
TYPE ST_Zone_Sensors :
STRUCT
    Temp_Room : REAL;
    Temp_Floor : REAL;
    Motion_Active : BOOL;
    Switch_Physical : BOOL;
    Light_State : BOOL;
    Maintenance : ST_Component_Maintenance;
END_STRUCT
END_TYPE

// GVL/GVL_BlackBox
{attribute 'qualified_only'}
VAR_GLOBAL
    // Буфер на 100 записей (при опросе 100мс это 10 секунд истории)
    G_BlackBox_Buffer : ARRAY[0..99] OF ST_BlackBox_Record;
    G_BlackBox_Frozen : BOOL;
    G_BlackBox_LastIndex : INT;
END_VAR

// GVL/GVL_Constants
{attribute 'qualified_only'}
VAR_GLOBAL CONSTANT
    C_MS_PER_SEC    : UDINT := 1000;
    C_SEC_PER_MIN   : UDINT := 60;
    C_MIN_PER_HOUR  : UDINT := 60;
    C_MS_PER_MIN    : UDINT := 60000;
    C_MAX_RULES     : INT := 20;
    C_ZONE_COUNT    : BYTE := 18;
END_VAR

// GVL/GVL_Diagnostics
{attribute 'qualified_only'}
VAR_GLOBAL
    G_Pump_Health : ARRAY[1..5] OF ST_Device_Health; // Для 5 коллекторных насосов
    G_Gas_Valve_Health : ST_Device_Health;
    G_System_Health_Summary : BYTE := 100;
END_VAR

// GVL/GVL_Global_Variables
{attribute 'qualified_only'}
VAR_GLOBAL
    GVL_System_Time_MS          : UDINT;
    GVL_IsActivePLC             : BOOL := TRUE;
    GVL_Local_PLC_Role          : E_PLC_ROLE := E_PLC_ROLE.ROLE_ACTIVE;
    
    // Данные датчиков
    GVL_Floor_Temps             : ARRAY[1..16] OF REAL;
    GVL_Valve_States            : ARRAY[1..3] OF BYTE;
END_VAR

// GVL/GVL_HMI_Config
VAR_GLOBAL
    // Настройки отопления (16 контуров)
    G_HMI_FloorHeating_Configs : ARRAY[1..16] OF ST_FloorHeating_Circuit_Config;
    G_HMI_Tariff_Settings : ST_Tariff_Config;
    
    // Настройки вентиляции (8 установок)
    G_HMI_Vent_Global_Config : ST_Ventilation_Global_Config;
    G_HMI_Vent_Unit_Configs : ARRAY[1..8] OF ST_Ventilation_Unit_Config;
    
    // Настройки освещения и сценариев
    G_HMI_Scenario_Configs : ARRAY[1..6] OF ST_Scenario_Config; // Для каждого типа сценария
    G_HMI_Outdoor_Configs : ARRAY[1..4] OF ST_Outdoor_Zone_Config;
    
    // Настройки безопасности
    G_HMI_Flood_Config : ST_Flood_Global_Config;
    G_HMI_Cleaning_Mode_Active : ARRAY[1..3] OF BOOL; // Режим уборки для 3-х зон протечки
    G_HMI_Cleaning_Mode_TimeLeft : ARRAY[1..3] OF UINT; // Оставшееся время (мин)
    G_HMI_Gas_Config : ST_Gas_Valve_Configuration;
    G_HMI_Admin_2FA_Enabled : BOOL := FALSE; // Настройка: 1 или 2 фактора для ADMIN
    G_HMI_Current_Operator_Factor2_Done : BOOL; // Флаг прохождения 2-го фактора
    
    // Калибровка датчиков (например, для 20 датчиков)
    G_HMI_Sensor_Calibrations : ARRAY[1..20] OF ST_Sensor_Calibration_Record;
    
    // Ручное управление клапанами с HMI (Override)
    G_HMI_Current_Operator_ID : STRING(10); // ID текущего авторизованного пользователя
    G_HMI_Manual_Gas_Valve_Open : BOOL; // Запрос на открытие
    G_HMI_Manual_Gas_Valve_Time : UDINT := 5; // Время в минутах
    G_HMI_Manual_Gas_Valve_TimeLeft : UDINT; // Оставшееся время (для вывода на HMI)
    
    // Команда на сохранение настроек в NVRAM
    G_HMI_Apply_Settings : BOOL;
    
    // Управление доступом (HMI)
    G_HMI_Gate_Open_Req : BOOL;
    G_HMI_Wicket_Open_Req : BOOL;
    G_HMI_Lock_1_Open_Req : BOOL;
    G_HMI_Lock_1_Close_Req : BOOL;
    G_HMI_Lock_2_Open_Req : BOOL;
    G_HMI_Lock_2_Close_Req : BOOL;
END_VAR

// GVL/GVL_IO
VAR_GLOBAL
    // Датчики открытия (15 физических каналов по ТЗ 3.1)
    DI_Security_Open : ARRAY[1..15] OF BOOL;
    
    // Датчики разбития (15 физических каналов по ТЗ 3.2)
    DI_Security_Glass : ARRAY[1..15] OF BOOL;
    
    // Групповой канал 2-го этажа
    DI_Security_2F_Group : BOOL;
    
    // Датчики протечки (12 штук по ТЗ 4.1)
    DI_Flood_Sensors : ARRAY[1..12] OF BOOL;
    
    // Смесительные узлы (5 коллекторов)
    AO_Manifold_Valves : ARRAY[1..5] OF UINT; // 0-1000 (Modbus)
    DO_Manifold_Pumps : ARRAY[1..5] OF BOOL;
    AI_Manifold_Currents : ARRAY[1..5] OF INT; // 4-20mA -> 400-2000
    AI_Manifold_Pressures : ARRAY[1..5] OF INT; // 0-10V -> 0-1000
    AI_Manifold_Temps_Supply : ARRAY[1..5] OF ST_Owen_Analog_Value;
    AI_Manifold_Temps_Return : ARRAY[1..5] OF INT;

    // Вентиляция
    AO_Supply_Fans : ARRAY[1..3] OF UINT; // 0-1000
    AO_Exhaust_Fans : ARRAY[1..5] OF UINT; // 0-1000
    
    // Котлы (BAXI Luna Platinum+ через OpenTherm)
    DO_Boiler_Enable : ARRAY[1..2] OF BOOL;
    AO_Boiler_Setpoint : ARRAY[1..2] OF UINT; // 0-1000 (0-100.0 C)
    AI_Boiler_Modulation : ARRAY[1..2] OF INT;
    AI_Boiler_Flame_Status : ARRAY[1..2] OF BOOL;
    DI_Boiler_Error : ARRAY[1..2] OF BOOL;
    
    // Газовые датчики (ТЗ 5.1, 5.2)
    AI_Methane_LEL : ARRAY[1..2] OF ST_Owen_Analog_Value; // 0-100% LEL
    AI_CO_PPM : ARRAY[1..8] OF REAL; // 0-1000 PPM
    DI_Smoke_Sensors : ARRAY[1..6] OF BOOL;
    
    // Аналоговые входы (AI)
    AI_Temp_Outdoor : ST_Owen_Analog_Value;
    AI_Floor_Temps : ARRAY[1..16] OF REAL;
    AI_Room_Temps : ARRAY[1..16] OF REAL; // Датчики температуры помещения (ТЗ 1.1)

    // Исполнительные механизмы ТП
    DO_Zone_Valves : ARRAY[1..16] OF BOOL; // Клапаны контуров ТП
    
    // ГВС (ТЗ 5.0)
    AI_DHW_Temp : REAL;
    AI_DHW_Pressure : REAL;
    DO_DHW_Heating_Pump : BOOL;
    DO_DHW_Circ_Pump : BOOL;
    
    // Освещение и Движение (ТЗ 1.0, 2.0)
    DI_Lighting_Switches : ARRAY[1..16] OF BOOL;
    DI_Motion_Sensors : ARRAY[1..16] OF BOOL;
    
    // Безопасность и Аварии
    DO_Gas_Valve_Close : BOOL;
    DO_Water_Valve_35_Close : BOOL;
    DO_Water_Valve_36_Close : BOOL;
    AI_Water_Valve_35_Current : REAL;
    AI_Water_Valve_36_Current : REAL;
    DI_Power_OK : BOOL;
    DO_Gas_Siren : BOOL;
    DO_Fire_Siren : BOOL;
    DO_Pump_Main_Enable : BOOL;
    
    // Управление доступом (Сухие контакты)
    DO_Gate_Open : BOOL;
    DO_Wicket_Open : BOOL;
    DO_Lock_1_Open : BOOL;
    DO_Lock_1_Close : BOOL;
    DO_Lock_2_Open : BOOL;
    DO_Lock_2_Close : BOOL;
END_VAR

// GVL/GVL_Vars
VAR_GLOBAL
    G_System_Time_MS : UDINT; // Системное время (мс)
    G_Current_Scenario : E_SCENARIO_TYPE := E_SCENARIO_TYPE.SCENARIO_NONE;
    G_Security_Armed : BOOL := FALSE;
    G_Gas_Alarm_Active : BOOL := FALSE;
    G_Fire_Alarm_Active : BOOL := FALSE;
    G_Flood_Alarm_Active : BOOL := FALSE;
    
    // Резервирование
    G_Local_PLC_ID : BYTE := 1; // ID текущего ПЛК (1 для A, 2 для B)
    G_Active_PLC_ID : BYTE := 1; // ID активного ПЛК в данный момент
    G_Remote_PLC_Pulse : BOOL; // Импульс от партнера
    
    // HMI и Конфигурация
    G_HMI_Current_Operator_ID : STRING(10) := 'ADMIN';
    G_HMI_Gas_Config : ST_Gas_Valve_Configuration;
    G_Heating_Config : ST_Heating_Config;
    G_Ventilation_Config : ST_Ventilation_Config;
    G_DHW_Config : ST_DHW_Config;
    G_Security_Config : ST_Security_Config;
    G_Flood_Config : ST_Flood_Config;
    G_HMI_Mute_Alarm : BOOL;
    G_HMI_Manual_Gas_Valve_Open : BOOL;
    G_HMI_Manual_Gas_Valve_Time : UDINT := 300000; // 5 минут по умолчанию
    G_HMI_Manual_Gas_Valve_TimeLeft : UDINT;
    
    // Состояние датчиков
    G_Floor_Temps : ARRAY[1..16] OF REAL;
    
    // Черный ящик
    G_BlackBox_Buffer : ARRAY[0..99] OF ST_BlackBox_Record;
    G_BlackBox_LastIndex : INT;
    G_BlackBox_Frozen : BOOL;
    
    // ТЗ 6.0: Обслуживание и ремонт
    G_Maintenance_Zones : ARRAY[1..16] OF ST_Component_Maintenance;
    G_Maintenance_Manifolds : ARRAY[1..5] OF ST_Component_Maintenance;
    G_Maintenance_Lighting : ARRAY[1..16] OF ST_Component_Maintenance;
    
    // Управление доступом (HMI)
    G_HMI_Gate_Open_Req : BOOL;
    G_HMI_Wicket_Open_Req : BOOL;
    G_HMI_Lock_1_Open_Req : BOOL;
    G_HMI_Lock_1_Close_Req : BOOL;
    G_HMI_Lock_2_Open_Req : BOOL;
    G_HMI_Lock_2_Close_Req : BOOL;
END_VAR

// PLC_A/Application/PRG_PLC_A
PROGRAM PRG_PLC_A
VAR
    L_PLC_ID : BYTE := 1;
END_VAR

// Установка глобального ID активного ПЛК (в реальной системе это определяется через механизм Heartbeat/Redundancy)
// Для ПЛК A: если он активен, G_Active_PLC_ID := 1
PRG_Main();

END_PROGRAM

// PRG_Main
PROGRAM PRG_Main
VAR
    // Менеджеры систем
    fbHeating : FB_Heating_System_Manager;
    fbSecurity : FB_Security_System_Manager;
    fbWater : FB_Water_Leakage_Manager;
    fbGasSmoke : FB_Gas_Smoke_Manager;
    fbVentilation : FB_Ventilation_System_Manager;
    fbRuleEngine : FB_User_Rule_Engine;
    fbLightingBlinds : FB_Lighting_Blinds_Manager;
    fbSimulation : FB_Simulation_Manager;
    fbDHW : FB_DHW_Manager; // ТЗ 5.0
    fbAccessControl : FB_Access_Control;
    
    // Системные блоки
    fbHeartbeat : FB_PLC_Heartbeat;
    fbNVRAM : FB_NVRAM_Manager;
    fbGateway : FB_Gateway_Interface;
    fbLogger : FB_Debug_Logger;
    
    // Локальные переменные
    L_Is_Active : BOOL;
    L_First_Cycle : BOOL := TRUE;
    L_System_State : ST_System_State_Summary;
    L_i : INT;
    L_Methane_LEL_Real : ARRAY[1..2] OF REAL;
    L_Manifold_Temps_Supply_Real : ARRAY[1..5] OF REAL;
    L_Manifold_Temps_Return_Real : ARRAY[1..5] OF REAL;
    L_Manifold_Pressures_Real : ARRAY[1..5] OF REAL;
    L_Manifold_Currents_Real : ARRAY[1..5] OF REAL;
    L_Current_TOD : TOD;
    
    // ТЗ 8.2: Распределение датчиков
    L_Opening_Sensors : ARRAY[1..15] OF BOOL;
    L_GlassBreak_Sensors : ARRAY[1..15] OF BOOL;
    L_Flood_Sensors : ARRAY[1..12] OF BOOL;
    
    L_Backup_Day : INT := 1; // ТЗ 16.2: Ротация 7 копий
END_VAR

// 0. Обновление системного времени
GVL_Vars.G_System_Time_MS := GVL_Vars.G_System_Time_MS + 10; 

// 1. Логика резервирования (ТЗ 11.1)
fbHeartbeat(
    VI_Local_ID := GVL_Vars.G_Local_PLC_ID,
    VI_System_Time := GVL_Vars.G_System_Time_MS,
    VI_Remote_Pulse := GVL_Vars.G_Remote_PLC_Pulse,
    VO_Is_Active => L_Is_Active
);
GVL_Vars.G_Active_PLC_ID := SEL(L_Is_Active, 0, GVL_Vars.G_Local_PLC_ID);

// 2. Инициализация и Бэкап (ТЗ 16.2)
L_Current_TOD := UDINT_TO_TOD(GVL_Vars.G_System_Time_MS MOD 86400000);
IF L_First_Cycle THEN
    L_First_Cycle := FALSE;
    fbNVRAM(VI_Command := 2, VI_RecordIndex := 1, VI_DataPtr := ADR(GVL_Vars.G_HMI_Gas_Config), VI_DataSize := SIZEOF(GVL_Vars.G_HMI_Gas_Config));
END_IF;

// Ежесуточный бэкап в 03:00 (ТЗ 16.2: Ротация 7 копий)
IF L_Current_TOD >= TOD#03:00 AND L_Current_TOD <= TOD#03:00:01 THEN
    fbNVRAM(VI_Command := 1, VI_RecordIndex := L_Backup_Day, VI_DataPtr := ADR(GVL_Vars.G_HMI_Gas_Config), VI_DataSize := SIZEOF(GVL_Vars.G_HMI_Gas_Config));
    L_Backup_Day := (L_Backup_Day MOD 7) + 1;
END_IF;

// 3. ТЗ 8.2: Параллельная обработка датчиков
FOR L_i := 1 TO 2 DO 
    L_Methane_LEL_Real[L_i] := GVL_IO.AI_Methane_LEL[L_i].rValue; 
END_FOR;
FOR L_i := 1 TO 5 DO 
    L_Manifold_Temps_Supply_Real[L_i] := GVL_IO.AI_Manifold_Temps_Supply[L_i].rValue; 
    L_Manifold_Temps_Return_Real[L_i] := TO_REAL(GVL_IO.AI_Manifold_Temps_Return[L_i]) / 10.0;
    L_Manifold_Pressures_Real[L_i] := TO_REAL(GVL_IO.AI_Manifold_Pressures[L_i]) / 100.0; // 0-10V -> 0-10.0 bar
    L_Manifold_Currents_Real[L_i] := TO_REAL(GVL_IO.AI_Manifold_Currents[L_i]) / 100.0; // 4-20mA -> 4.0-20.0 mA
END_FOR;

FOR L_i := 1 TO 15 DO
    // ПЛК A (ID=1) обрабатывает нечетные, ПЛК B (ID=2) - четные
    IF (GVL_Vars.G_Local_PLC_ID = 1 AND (L_i MOD 2 <> 0)) OR (GVL_Vars.G_Local_PLC_ID = 2 AND (L_i MOD 2 = 0)) THEN
        L_Opening_Sensors[L_i] := GVL_IO.DI_Security_Open[L_i];
        L_GlassBreak_Sensors[L_i] := GVL_IO.DI_Security_Glass[L_i];
    END_IF;
END_FOR;

FOR L_i := 1 TO 12 DO
    IF (GVL_Vars.G_Local_PLC_ID = 1 AND (L_i MOD 2 <> 0)) OR (GVL_Vars.G_Local_PLC_ID = 2 AND (L_i MOD 2 = 0)) THEN
        L_Flood_Sensors[L_i] := GVL_IO.DI_Flood_Sensors[L_i];
    END_IF;
END_FOR;

    // 4. Сбор состояния
    L_System_State.Outdoor_Temp := GVL_IO.AI_Temp_Outdoor.rValue;
    FOR L_i := 1 TO 16 DO 
        L_System_State.Floor_Temps[L_i] := GVL_IO.AI_Floor_Temps[L_i]; 
        L_System_State.Indoor_Temp[L_i] := GVL_IO.AI_Room_Temps[L_i];
        L_System_State.CO2[MIN(L_i, 8)] := 400.0; 
        L_System_State.Humidity[MIN(L_i, 8)] := 45.0; 
    END_FOR;
    L_System_State.Security_Armed := GVL_Vars.G_Security_Armed;
    L_System_State.Flood_Alarm := GVL_Vars.G_Flood_Alarm_Active;
    L_System_State.Gas_Alarm := GVL_Vars.G_Gas_Alarm_Active;
    L_System_State.Fire_Alarm := GVL_Vars.G_Fire_Alarm_Active;

    // 5. Выполнение системной логики
    fbGasSmoke(
        VI_System_Time_MS := GVL_Vars.G_System_Time_MS,
        VI_IsActivePLC := L_Is_Active,
        VI_Methane_LEL := L_Methane_LEL_Real,
        VI_CO_PPM := GVL_IO.AI_CO_PPM,
        VI_Smoke_Sensors := GVL_IO.DI_Smoke_Sensors,
        VI_Mute_Request := GVL_Vars.G_HMI_Mute_Alarm,
        VO_Gas_Alarm => GVL_Vars.G_Gas_Alarm_Active,
        VO_Fire_Alarm => GVL_Vars.G_Fire_Alarm_Active,
        VO_Gas_Valve_Close => GVL_IO.DO_Gas_Valve_Close
    );

    // ТЗ 3.6: При тревоге -> долгосрочный отъезд
    IF fbSecurity.VO_Long_Away_Req THEN
        GVL_Vars.G_Current_Scenario := E_SCENARIO_TYPE.SCENARIO_AWAY;
    END_IF;

    fbWater(
        VI_System_Time_MS := GVL_Vars.G_System_Time_MS,
        VI_IsActivePLC := L_Is_Active,
        VI_Sensors := L_Flood_Sensors,
        VI_Valve_35_Current := GVL_IO.AI_Water_Valve_35_Current,
        VI_Valve_36_Current := GVL_IO.AI_Water_Valve_36_Current,
        VI_Config := GVL_Vars.G_Flood_Config,
        VI_Power_OK := GVL_IO.DI_Power_OK,
        VO_Flood_Alarm => GVL_Vars.G_Flood_Alarm_Active,
        VO_Valve_35_Close => GVL_IO.DO_Water_Valve_35_Close,
        VO_Valve_36_Close => GVL_IO.DO_Water_Valve_36_Close
    );

    fbHeating(
        VI_System_Time_MS := GVL_Vars.G_System_Time_MS,
        VI_IsActivePLC := L_Is_Active AND NOT fbGasSmoke.VO_Boiler_Stop,
        VI_Outdoor_Temp := L_System_State.Outdoor_Temp,
        VI_Floor_Temps := GVL_IO.AI_Floor_Temps,
        VI_Room_Temps := GVL_IO.AI_Room_Temps,
        VI_Config := GVL_Vars.G_Heating_Config,
        VI_Manifold_Temps_Supply := L_Manifold_Temps_Supply_Real,
        VI_Manifold_Temps_Return := L_Manifold_Temps_Return_Real,
        VI_Manifold_Pressures := L_Manifold_Pressures_Real,
        VI_Manifold_Currents := L_Manifold_Currents_Real,
        VI_Boiler_Flame_Status := GVL_IO.AI_Boiler_Flame_Status,
        VI_Maintenance_Zones := GVL_Vars.G_Maintenance_Zones,
        VI_Maintenance_Manifolds := GVL_Vars.G_Maintenance_Manifolds,
        VO_Manifold_Pumps => GVL_IO.DO_Manifold_Pumps,
        VO_Zone_Valves => GVL_IO.DO_Zone_Valves,
        VO_Boiler_Enable => GVL_IO.DO_Boiler_Enable
    );
    // Конверсия выходов для Modbus
    FOR L_i := 1 TO 5 DO GVL_IO.AO_Manifold_Valves[L_i] := TO_UINT(fbHeating.VO_Manifold_Valves[L_i] * 10.0); END_FOR;
    FOR L_i := 1 TO 2 DO GVL_IO.AO_Boiler_Setpoint[L_i] := TO_UINT(fbHeating.VO_Boiler_Setpoint[L_i] * 10.0); END_FOR;

fbSecurity(
    VI_System_Time_MS := GVL_Vars.G_System_Time_MS,
    VI_IsActivePLC := L_Is_Active,
    VI_Opening_Sensors := L_Opening_Sensors,
    VI_GlassBreak_Sensors := L_GlassBreak_Sensors,
    VI_Config := GVL_Vars.G_Security_Config,
    VI_Group_2F_Open := GVL_IO.DI_Security_2F_Group, // ТЗ 3.1
    VI_Group_2F_Glass := GVL_IO.DI_Security_2F_Group, // ТЗ 3.2 (используем тот же канал если не выделен)
    VO_Armed => GVL_Vars.G_Security_Armed
);

fbAccessControl(
    VI_System_Time_MS := GVL_Vars.G_System_Time_MS,
    VI_IsActivePLC := L_Is_Active,
    VI_Armed := GVL_Vars.G_Security_Armed,
    VI_Gate_Open_Req := GVL_Vars.G_HMI_Gate_Open_Req,
    VI_Wicket_Open_Req := GVL_Vars.G_HMI_Wicket_Open_Req,
    VI_Lock_1_Open_Req := GVL_Vars.G_HMI_Lock_1_Open_Req,
    VI_Lock_1_Close_Req := GVL_Vars.G_HMI_Lock_1_Close_Req,
    VI_Lock_2_Open_Req := GVL_Vars.G_HMI_Lock_2_Open_Req,
    VI_Lock_2_Close_Req := GVL_Vars.G_HMI_Lock_2_Close_Req,
    VI_Config := GVL_Vars.G_Security_Config
);

// Сброс команд HMI (импульсные кнопки)
IF GVL_Vars.G_HMI_Gate_Open_Req AND NOT fbAccessControl.VO_Gate_Open THEN GVL_Vars.G_HMI_Gate_Open_Req := FALSE; END_IF;
IF GVL_Vars.G_HMI_Wicket_Open_Req AND NOT fbAccessControl.VO_Wicket_Open THEN GVL_Vars.G_HMI_Wicket_Open_Req := FALSE; END_IF;
IF GVL_Vars.G_HMI_Lock_1_Open_Req AND NOT fbAccessControl.VO_Lock_1_Open THEN GVL_Vars.G_HMI_Lock_1_Open_Req := FALSE; END_IF;
IF GVL_Vars.G_HMI_Lock_1_Close_Req AND NOT fbAccessControl.VO_Lock_1_Close THEN GVL_Vars.G_HMI_Lock_1_Close_Req := FALSE; END_IF;
IF GVL_Vars.G_HMI_Lock_2_Open_Req AND NOT fbAccessControl.VO_Lock_2_Open THEN GVL_Vars.G_HMI_Lock_2_Open_Req := FALSE; END_IF;
IF GVL_Vars.G_HMI_Lock_2_Close_Req AND NOT fbAccessControl.VO_Lock_2_Close THEN GVL_Vars.G_HMI_Lock_2_Close_Req := FALSE; END_IF;

// Маппинг на физические выходы
GVL_IO.DO_Gate_Open := fbAccessControl.VO_Gate_Open;
GVL_IO.DO_Wicket_Open := fbAccessControl.VO_Wicket_Open;
GVL_IO.DO_Lock_1_Open := fbAccessControl.VO_Lock_1_Open;
GVL_IO.DO_Lock_1_Close := fbAccessControl.VO_Lock_1_Close;
GVL_IO.DO_Lock_2_Open := fbAccessControl.VO_Lock_2_Open;
GVL_IO.DO_Lock_2_Close := fbAccessControl.VO_Lock_2_Close;

fbDHW(
    VI_System_Time_MS := GVL_Vars.G_System_Time_MS,
    VI_IsActivePLC := L_Is_Active,
    VI_Temp := GVL_IO.AI_DHW_Temp,
    VI_Pressure := GVL_IO.AI_DHW_Pressure,
    VI_Config := GVL_Vars.G_DHW_Config,
    VI_Maintenance := GVL_Vars.G_Maintenance_Lighting[1] // Условно используем ячейку для ГВС
);
GVL_IO.DO_DHW_Heating_Pump := fbDHW.VO_Heating_Pump;
GVL_IO.DO_DHW_Circ_Pump := fbDHW.VO_Circ_Pump;

fbVentilation(
    VI_System_Time_MS := GVL_Vars.G_System_Time_MS,
    VI_IsActivePLC := L_Is_Active,
    VI_CO2 := L_System_State.CO2,
    VI_Humidity := L_System_State.Humidity,
    VI_Gas_Alarm := GVL_Vars.G_Gas_Alarm_Active,
    VI_Fire_Alarm := GVL_Vars.G_Fire_Alarm_Active,
    VI_Flood_Alarm := GVL_Vars.G_Flood_Alarm_Active,
    VI_Config := GVL_Vars.G_Ventilation_Config,
    VI_PV3_Boost := fbGasSmoke.VO_Vent_PV3_Boost, // ТЗ 5.1
    VI_Supply_100_Req := fbGasSmoke.VO_Supply_100_Req, // ТЗ 6.4
    VI_Exhaust_100_Req := fbGasSmoke.VO_Exhaust_100_Req, // ТЗ 6.4
    VI_Supply_80_Req := fbGasSmoke.VO_Supply_80_Req, // ТЗ 5.4
    VI_Wet_Zone_Lights := fbLightingBlinds.VO_Wet_Zone_Light_Active // ТЗ 4.0
);
// Конверсия выходов вентиляции
FOR L_i := 1 TO 3 DO GVL_IO.AO_Supply_Fans[L_i] := TO_UINT(fbVentilation.VO_Supply_Fans[L_i] * 10.0); END_FOR;
FOR L_i := 1 TO 5 DO GVL_IO.AO_Exhaust_Fans[L_i] := TO_UINT(fbVentilation.VO_Exhaust_Fans[L_i] * 10.0); END_FOR;

fbSimulation(
    VI_System_Time_MS := GVL_Vars.G_System_Time_MS,
    VI_Enabled := (GVL_Vars.G_Current_Scenario = E_SCENARIO_TYPE.SCENARIO_AWAY),
    VI_Intensity := 0.3
);

fbLightingBlinds(
    VI_System_Time_MS := GVL_Vars.G_System_Time_MS,
    VI_IsActivePLC := L_Is_Active,
    VI_Current_Scenario := GVL_Vars.G_Current_Scenario,
    VI_Away_Level := fbSecurity.VO_Away_Level,
    VI_Simulation_Active := (GVL_Vars.G_Current_Scenario = E_SCENARIO_TYPE.SCENARIO_AWAY),
    VI_Simulation_Lights := fbSimulation.VO_Light_States,
    VI_Physical_Switches := GVL_IO.DI_Lighting_Switches, // ТЗ 1.0
    VI_Motion_Sensors := GVL_IO.DI_Motion_Sensors, // ТЗ 2.0
    VI_Maintenance := GVL_Vars.G_Maintenance_Lighting // ТЗ 6.0
);

fbRuleEngine(VI_System_State := L_System_State);

fbGateway(
    VI_System_Time_MS := GVL_Vars.G_System_Time_MS,
    VI_Local_PLC_Role := SEL(L_Is_Active, E_PLC_ROLE.ROLE_STANDBY, E_PLC_ROLE.ROLE_ACTIVE),
    VI_FloorHeating_Temps := GVL_IO.AI_Floor_Temps,
    VI_Room_Temps := GVL_IO.AI_Room_Temps,
    VI_Zone_Valve_States := GVL_IO.DO_Zone_Valves,
    VI_Manifold_Pressures := L_Manifold_Pressures_Real,
    VI_Manifold_Pump_States := GVL_IO.DO_Manifold_Pumps,
    VI_Outdoor_Temp := L_System_State.Outdoor_Temp,
    VI_Security_Armed := GVL_Vars.G_Security_Armed,
    VI_Flood_Alarm_Active := GVL_Vars.G_Flood_Alarm_Active,
    VI_Gas_Alarm_Active := GVL_Vars.G_Gas_Alarm_Active,
    VI_Fire_Alarm_Active := GVL_Vars.G_Fire_Alarm_Active,
    VI_Lighting_Base_Levels := fbLightingBlinds.VO_Lighting_Levels,
    VI_Blinds_Positions := fbLightingBlinds.VO_Blinds_Positions,
    VI_Active_Scenario := GVL_Vars.G_Current_Scenario
);

END_PROGRAM

// POUs/FB_Heating_System_Manager
FUNCTION_BLOCK FB_Heating_System_Manager
VAR_INPUT
    VI_Maintenance_Zones : ARRAY[1..16] OF ST_Component_Maintenance;
    VI_Maintenance_Manifolds : ARRAY[1..5] OF ST_Component_Maintenance;
    VI_System_Time_MS : UDINT;
    VI_IsActivePLC : BOOL;
    VI_Outdoor_Temp : REAL;
    VI_Floor_Temps : ARRAY[1..16] OF REAL;
    VI_Room_Temps : ARRAY[1..16] OF REAL;
    VI_Config : ST_Heating_Config;
    VI_Manifold_Pressures : ARRAY[1..5] OF REAL;
    VI_Manifold_Currents : ARRAY[1..5] OF REAL;
    VI_Manifold_Temps_Supply : ARRAY[1..5] OF REAL;
    VI_Manifold_Temps_Return : ARRAY[1..5] OF REAL;
    VI_Boiler_Flame_Status : ARRAY[1..2] OF BOOL;
END_VAR
VAR_OUTPUT
    VO_Manifold_Valves : ARRAY[1..5] OF REAL; // 0-100%
    VO_Manifold_Pumps : ARRAY[1..5] OF BOOL;
    VO_Zone_Valves : ARRAY[1..16] OF BOOL;
    VO_Boiler_Enable : ARRAY[1..2] OF BOOL;
    VO_Boiler_Setpoint : ARRAY[1..2] OF REAL; // OpenTherm Setpoint
    VO_Status : ARRAY[1..5] OF ST_Manifold_Status;
    VO_Boiler_Status : ARRAY[1..2] OF ST_Boiler_Status;
END_VAR
VAR
    L_PID_Valves : ARRAY[1..5] OF FB_PID_Controller;
    L_Last_Boiler_Rotation : UDINT;
    L_Lead_Boiler : BYTE := 1;
    L_i : INT;
    L_Target_Supply_Temp : REAL;
    L_Demand_Power : REAL;
    L_Any_Zone_Active : ARRAY[1..5] OF BOOL;
    
    // ТЗ 2.5: Задержка перегрева
    L_Overheat_Timer : ARRAY[1..16] OF TON;
    
    // ТЗ 2.6: Диагностика
    L_Pump_Run_Timer : ARRAY[1..5] OF TON;
    L_Pump_Pause_Timer : ARRAY[1..5] OF TON;
    L_Pump_In_Pause : ARRAY[1..5] OF BOOL;
    
    // ТЗ 2.8: Учет наработки
    L_Last_Scan_Time : UDINT;
    L_Lifespan_S : REAL := 180000000.0; // 50,000 hours in seconds
END_VAR

// 1. Расчет целевой температуры подачи (ТЗ 2.3)
L_Target_Supply_Temp := 35.0;
IF VI_Config.Weather_Comp_Enabled AND VI_Outdoor_Temp < 15.0 THEN
    // Исправлено: убран множитель 10.0 согласно ТЗ 2.3
    L_Target_Supply_Temp := L_Target_Supply_Temp + (15.0 - VI_Outdoor_Temp) * VI_Config.Weather_Coef;
END_IF;
L_Target_Supply_Temp := LIMIT(20.0, L_Target_Supply_Temp, 45.0);

// 2. Управление зонами (ТЗ 1.1, 2.5)
FOR L_i := 1 TO 16 DO
    L_Overheat_Timer[L_i](IN := VI_Floor_Temps[L_i] > VI_Config.Overheat_Threshold, PT := T#60s);
    
    IF VI_Room_Temps[L_i] < (VI_Config.Target_Room_Temp - VI_Config.Hysteresis) THEN
        VO_Zone_Valves[L_i] := TRUE;
    ELSIF VI_Room_Temps[L_i] > (VI_Config.Target_Room_Temp + VI_Config.Hysteresis) THEN
        VO_Zone_Valves[L_i] := FALSE;
    END_IF;
    
    // Защита от перегрева с задержкой 60с (ТЗ 2.5)
    IF L_Overheat_Timer[L_i].Q THEN
        VO_Zone_Valves[L_i] := FALSE;
    END_IF;
END_FOR;

// 3. Активность коллекторов
L_Any_Zone_Active[1] := VO_Zone_Valves[1] OR VO_Zone_Valves[2];
L_Any_Zone_Active[2] := VO_Zone_Valves[3] OR VO_Zone_Valves[4] OR VO_Zone_Valves[5] OR VO_Zone_Valves[6];
L_Any_Zone_Active[3] := VO_Zone_Valves[7] OR VO_Zone_Valves[8] OR VO_Zone_Valves[9];
L_Any_Zone_Active[4] := VO_Zone_Valves[10] OR VO_Zone_Valves[11] OR VO_Zone_Valves[12];
L_Any_Zone_Active[5] := VO_Zone_Valves[13] OR VO_Zone_Valves[14] OR VO_Zone_Valves[15] OR VO_Zone_Valves[16];

// 4. Управление коллекторами (ТЗ 2.6, 12.2)
FOR L_i := 1 TO 5 DO
    L_PID_Valves[L_i](
        VI_SetPoint := L_Target_Supply_Temp,
        VI_ProcessValue := VI_Manifold_Temps_Supply[L_i],
        VI_Kp := 2.0, VI_Tn := 120.0, VI_Tv := 0.0,
        VI_Y_Min := 0.0, VI_Y_Max := 100.0, VI_Cycle_Time_S := 1.0,
        VO_Output => VO_Manifold_Valves[L_i]
    );

    // ТЗ 2.6: Пауза после 72 часов работы
    L_Pump_Run_Timer[L_i](IN := VO_Manifold_Pumps[L_i] AND NOT L_Pump_In_Pause[L_i], PT := T#72h);
    IF L_Pump_Run_Timer[L_i].Q THEN L_Pump_In_Pause[L_i] := TRUE; END_IF;
    
    L_Pump_Pause_Timer[L_i](IN := L_Pump_In_Pause[L_i], PT := T#1h);
    IF L_Pump_Pause_Timer[L_i].Q THEN L_Pump_In_Pause[L_i] := FALSE; END_IF;

    VO_Manifold_Pumps[L_i] := VI_IsActivePLC AND L_Any_Zone_Active[L_i] AND NOT L_Pump_In_Pause[L_i];

    // Защита от замерзания (ТЗ 2.4)
    IF VI_Outdoor_Temp < -5.0 OR VI_Manifold_Temps_Supply[L_i] < VI_Config.Freeze_Threshold THEN
        VO_Manifold_Pumps[L_i] := TRUE;
        VO_Manifold_Valves[L_i] := 100.0;
    END_IF;

    // Диагностика (ТЗ 2.6)
    VO_Status[L_i].Pump_On := VO_Manifold_Pumps[L_i];
    VO_Status[L_i].Pump_Current := VI_Manifold_Currents[L_i];
    VO_Status[L_i].Pressure := VI_Manifold_Pressures[L_i];
    VO_Status[L_i].Temp_Supply := VI_Manifold_Temps_Supply[L_i];
    VO_Status[L_i].Temp_Return := VI_Manifold_Temps_Return[L_i];
    VO_Status[L_i].Valve_Pos := VO_Manifold_Valves[L_i];
    
    // Контроль давления (1.5-2.5 бар) и Delta T (5-10C)
    IF VO_Manifold_Pumps[L_i] THEN
        IF VI_Manifold_Pressures[L_i] < 1.5 OR VI_Manifold_Pressures[L_i] > 2.5 THEN
            VO_Status[L_i].Error := TRUE; VO_Status[L_i].Error_ID := 16#E004; // Pressure Out of Range
        END_IF;
        // Исправлено: порог Delta T снижен до 10.0 согласно ТЗ 2.6
        IF (VI_Manifold_Temps_Supply[L_i] - VI_Manifold_Temps_Return[L_i]) > 10.0 THEN
            VO_Status[L_i].Error := TRUE; VO_Status[L_i].Error_ID := 16#E005; // High Delta T
        END_IF;
    END_IF;

    // Тестирование арматуры (ТЗ 12.2)
    IF (VI_System_Time_MS MOD 604800000) < 10000 THEN VO_Manifold_Valves[L_i] := 20.0; END_IF;
END_FOR;

// 5. Каскад котлов (ТЗ 2.8, 12.3)
L_Demand_Power := 0.0;
FOR L_i := 1 TO 5 DO IF VO_Manifold_Pumps[L_i] THEN L_Demand_Power := L_Demand_Power + VO_Manifold_Valves[L_i]; END_IF; END_FOR;
L_Demand_Power := L_Demand_Power / 5.0;

IF (VI_System_Time_MS - L_Last_Boiler_Rotation) > 604800000 THEN
    L_Last_Boiler_Rotation := VI_System_Time_MS;
    L_Lead_Boiler := SEL(L_Lead_Boiler = 1, 1, 2);
END_IF;

IF VI_IsActivePLC AND L_Demand_Power > 5.0 THEN
    VO_Boiler_Enable[L_Lead_Boiler] := TRUE;
    VO_Boiler_Setpoint[L_Lead_Boiler] := L_Target_Supply_Temp + 5.0; // OpenTherm Setpoint
    VO_Boiler_Enable[3 - L_Lead_Boiler] := (L_Demand_Power > 80.0);
    VO_Boiler_Setpoint[3 - L_Lead_Boiler] := SEL(L_Demand_Power > 80.0, 0.0, L_Target_Supply_Temp + 5.0);
ELSE
    VO_Boiler_Enable[1] := FALSE; VO_Boiler_Enable[2] := FALSE;
END_IF;

// Учет наработки (ТЗ 2.8, 12.3)
FOR L_i := 1 TO 2 DO
    IF VI_Boiler_Flame_Status[L_i] THEN
        VO_Boiler_Status[L_i].Work_Seconds := VO_Boiler_Status[L_i].Work_Seconds + 1; // Assuming 1s cycle for this FB or call
        VO_Boiler_Status[L_i].Work_Hours := TO_REAL(VO_Boiler_Status[L_i].Work_Seconds) / 3600.0;
        VO_Boiler_Status[L_i].Resource_Percent := (1.0 - (TO_REAL(VO_Boiler_Status[L_i].Work_Seconds) / L_Lifespan_S)) * 100.0;
    END_IF;
    VO_Boiler_Status[L_i].Running := VI_Boiler_Flame_Status[L_i];
END_FOR;

END_FUNCTION_BLOCK

// POUs/FB_PID_Controller
FUNCTION_BLOCK FB_PID_Controller
VAR_INPUT
    VI_SetPoint : REAL;         // Уставка
    VI_ProcessValue : REAL;     // Текущее значение
    VI_Kp : REAL;               // Коэффициент усиления
    VI_Tn : REAL;               // Время интегрирования (сек)
    VI_Tv : REAL;               // Время дифференцирования (сек)
    VI_Y_Min : REAL := 0.0;     // Минимальный выход
    VI_Y_Max : REAL := 100.0;   // Максимальный выход
    VI_Manual_Mode : BOOL;      // Ручной режим
    VI_Manual_Value : REAL;     // Значение в ручном режиме
    VI_Deadband : REAL := 0.1;  // Мертвая зона
    VI_Cycle_Time_S : REAL := 0.01; // Время цикла задачи в секундах
    VI_Reset : BOOL;            // Сброс интегральной составляющей
END_VAR
VAR_OUTPUT
    VO_Output : REAL;           // Выход регулятора
    VO_Error : REAL;            // Ошибка рассогласования
    VO_Limiting : BOOL;         // Флаг ограничения выхода (Anti-windup)
END_VAR
VAR
    L_Integral_Sum : REAL;      // Интегральная сумма
    L_Prev_Error : REAL;        // Предыдущая ошибка
    L_Derivative : REAL;        // Дифференциальная составляющая
    L_Output_Raw : REAL;        // Сырой выход до ограничения
END_VAR

// Расчет ошибки
VO_Error := VI_SetPoint - VI_ProcessValue;

// Проверка мертвой зоны
IF ABS(VO_Error) < VI_Deadband THEN
    VO_Error := 0.0;
END_IF;

IF VI_Reset THEN
    L_Integral_Sum := 0.0;
    L_Prev_Error := 0.0;
    VO_Output := 0.0;
    RETURN;
END_IF;

IF VI_Manual_Mode THEN
    VO_Output := VI_Manual_Value;
    L_Integral_Sum := VO_Output; // Безударный переход
    RETURN;
END_IF;

// Пропорциональная составляющая
L_Output_Raw := VI_Kp * VO_Error;

// Интегральная составляющая (Метод трапеций)
IF VI_Tn > 0.0 THEN
    // Anti-windup: не накапливаем интеграл, если выход уже на пределе и ошибка того же знака
    IF NOT VO_Limiting OR (VO_Error > 0.0 AND L_Output_Raw < VI_Y_Max) OR (VO_Error < 0.0 AND L_Output_Raw > VI_Y_Min) THEN
        L_Integral_Sum := L_Integral_Sum + (VI_Kp / VI_Tn) * VO_Error * VI_Cycle_Time_S;
    END_IF;
    L_Output_Raw := L_Output_Raw + L_Integral_Sum;
END_IF;

// Дифференциальная составляющая
IF VI_Tv > 0.0 THEN
    L_Derivative := (VO_Error - L_Prev_Error) / VI_Cycle_Time_S;
    L_Output_Raw := L_Output_Raw + VI_Kp * VI_Tv * L_Derivative;
END_IF;

L_Prev_Error := VO_Error;

// Ограничение выхода
IF L_Output_Raw > VI_Y_Max THEN
    VO_Output := VI_Y_Max;
    VO_Limiting := TRUE;
ELSIF L_Output_Raw < VI_Y_Min THEN
    VO_Output := VI_Y_Min;
    VO_Limiting := TRUE;
ELSE
    VO_Output := L_Output_Raw;
    VO_Limiting := FALSE;
END_IF;

END_FUNCTION_BLOCK

// POUs/FB_Security_System_Manager
FUNCTION_BLOCK FB_Security_System_Manager
VAR_INPUT
    VI_System_Time_MS : UDINT;
    VI_IsActivePLC : BOOL;
    VI_Opening_Sensors : ARRAY[1..15] OF BOOL;
    VI_GlassBreak_Sensors : ARRAY[1..15] OF BOOL;
    VI_PIN_Input : STRING(4);
    VI_PIN_Submit : BOOL;
    VI_Config : ST_Security_Config;
    VI_Outdoor_Lux : REAL;
    VI_Motion_Corridor : BOOL;
    VI_Acknowledge_Open_Windows : BOOL; // ТЗ 3.8
    VI_Group_2F_Open : BOOL; // ТЗ 3.1 (7 окон -> 1 канал)
    VI_Group_2F_Glass : BOOL; // ТЗ 3.2
END_VAR
VAR_OUTPUT
    VO_Armed : BOOL;
    VO_Alarm_Active : BOOL;
    VO_Entry_Delay_Active : BOOL;
    VO_Time_To_Alarm_S : UINT;
    VO_Away_Level : BYTE; // 1-Short, 2-Medium, 3-Long
    VO_Light_Corridor : BOOL;
    VO_Light_Stairs_Dim : BYTE;
    VO_Status_Msg : STRING(200);
    VO_Long_Away_Req : BOOL; // ТЗ 3.6: При тревоге -> долгосрочный отъезд
END_VAR
VAR
    L_State : BYTE; // 0-Disarmed, 1-Armed, 2-EntryDelay, 3-Alarm, 4-ConfirmWait
    L_Attempts : UINT;
    L_Entry_Start_Time : UDINT;
    L_Away_Start_Time : UDINT;
    L_Confirm_Start_Time : UDINT;
    L_Last_Trigger_Time : UDINT;
    L_i : INT;
    L_Any_Sensor_Open : BOOL;
    L_Any_Glass_Broken : BOOL;
    
    // ТЗ 3.3: Комбинированные события (>=2 за 10с)
    L_Trigger_Count : UINT;
    L_Trigger_Timer : TON;
    L_Last_Sensors : ARRAY[1..32] OF BOOL;
    
    // ТЗ 3.8: Снижение порога
    L_Glass_Threshold_Multiplier : REAL := 1.0;
END_VAR

// 1. Мониторинг датчиков
L_Any_Sensor_Open := VI_Group_2F_Open;
FOR L_i := 1 TO 15 DO IF VI_Opening_Sensors[L_i] THEN L_Any_Sensor_Open := TRUE; EXIT; END_IF; END_FOR;

L_Any_Glass_Broken := VI_Group_2F_Glass;
FOR L_i := 1 TO 15 DO IF VI_GlassBreak_Sensors[L_i] THEN L_Any_Glass_Broken := TRUE; EXIT; END_IF; END_FOR;

// ТЗ 3.3: Подсчет срабатываний за 10с
L_Trigger_Timer(IN := L_Trigger_Count > 0, PT := T#10s);
IF L_Trigger_Timer.Q THEN L_Trigger_Count := 0; END_IF;

FOR L_i := 1 TO 15 DO
    IF VI_Opening_Sensors[L_i] AND NOT L_Last_Sensors[L_i] THEN L_Trigger_Count := L_Trigger_Count + 1; END_IF;
    L_Last_Sensors[L_i] := VI_Opening_Sensors[L_i];
    
    IF VI_GlassBreak_Sensors[L_i] AND NOT L_Last_Sensors[15 + L_i] THEN L_Trigger_Count := L_Trigger_Count + 1; END_IF;
    L_Last_Sensors[15 + L_i] := VI_GlassBreak_Sensors[L_i];
END_FOR;
// Групповые датчики тоже участвуют в подсчете
IF VI_Group_2F_Open AND NOT L_Last_Sensors[31] THEN L_Trigger_Count := L_Trigger_Count + 1; END_IF;
L_Last_Sensors[31] := VI_Group_2F_Open;
IF VI_Group_2F_Glass AND NOT L_Last_Sensors[32] THEN L_Trigger_Count := L_Trigger_Count + 1; END_IF;
L_Last_Sensors[32] := VI_Group_2F_Glass;

// ТЗ 3.8: Снижение порога на 20% (увеличиваем чувствительность)
L_Glass_Threshold_Multiplier := SEL(VI_Acknowledge_Open_Windows, 1.0, 0.8);

// 2. Логика состояний
CASE L_State OF
    0: // Снято с охраны
        VO_Armed := FALSE; VO_Alarm_Active := FALSE; VO_Entry_Delay_Active := FALSE; VO_Long_Away_Req := FALSE;
        IF VI_PIN_Submit AND VI_PIN_Input = VI_Config.PIN_Code THEN
            IF NOT L_Any_Sensor_Open OR VI_Acknowledge_Open_Windows THEN
                IF VI_Config.Two_Stage_Mode THEN
                    L_State := 4; L_Confirm_Start_Time := VI_System_Time_MS;
                    VO_Status_Msg := 'Ожидание второго этапа подтверждения';
                ELSE
                    L_State := 1; L_Away_Start_Time := VI_System_Time_MS; L_Attempts := 0;
                    VO_Status_Msg := 'Система поставлена на охрану';
                END_IF;
            ELSE
                VO_Status_Msg := 'Ошибка: Обнаружены открытые окна/двери';
            END_IF;
        END_IF;

    4: // Ожидание второго этапа (ТЗ 3.4)
        IF (VI_System_Time_MS - L_Confirm_Start_Time) / 1000 >= VI_Config.Confirmation_Timeout_S THEN
            L_State := 0; VO_Status_Msg := 'Таймаут подтверждения постановки';
        ELSIF VI_PIN_Submit AND VI_PIN_Input = VI_Config.PIN_Code THEN
             L_State := 1; L_Away_Start_Time := VI_System_Time_MS; L_Attempts := 0;
             VO_Status_Msg := 'Система поставлена на охрану (2 этапа)';
        END_IF;

    1: // На охране
        VO_Armed := TRUE;
        // ТЗ 3.3: Немедленная тревога если >=2 датчика за 10с
        IF L_Trigger_Count >= 2 THEN
            L_State := 3;
        ELSIF L_Any_Sensor_Open OR L_Any_Glass_Broken THEN
            L_State := 2; L_Entry_Start_Time := VI_System_Time_MS;
        END_IF;

    2: // Задержка входа (ТЗ 3.3)
        VO_Entry_Delay_Active := TRUE;
        VO_Time_To_Alarm_S := TO_UINT(VI_Config.Entry_Delay_S - (VI_System_Time_MS - L_Entry_Start_Time) / 1000);
        IF VI_PIN_Submit THEN
            IF VI_PIN_Input = VI_Config.PIN_Code THEN L_State := 0; VO_Status_Msg := 'Система снята с охраны';
            ELSE
                L_Attempts := L_Attempts + 1;
                IF L_Attempts >= VI_Config.Max_Attempts THEN L_State := 3; END_IF;
            END_IF;
        END_IF;
        IF (VI_System_Time_MS - L_Entry_Start_Time) / 1000 >= VI_Config.Entry_Delay_S THEN L_State := 3; END_IF;

    3: // Тревога
        VO_Alarm_Active := TRUE;
        VO_Long_Away_Req := TRUE; // ТЗ 3.6: При тревоге -> долгосрочный отъезд
        VO_Status_Msg := 'ТРЕВОГА: НАРУШЕНИЕ ПЕРИМЕТРА';
        IF VI_PIN_Submit AND VI_PIN_Input = VI_Config.PIN_Code THEN L_State := 0; VO_Status_Msg := 'Тревога сброшена'; END_IF;
END_CASE;

// 3. Уровни отъезда (ТЗ 3.5)
IF L_State <> 0 THEN
    L_Last_Trigger_Time := (VI_System_Time_MS - L_Away_Start_Time) / 3600000; // Часы
    IF L_Last_Trigger_Time < 2 THEN VO_Away_Level := 1;
    ELSIF L_Last_Trigger_Time < 72 THEN VO_Away_Level := 2;
    ELSE VO_Away_Level := 3; END_IF;
ELSE VO_Away_Level := 0; END_IF;

// 4. Интеграция с освещением (ТЗ 3.9)
IF (VI_Outdoor_Lux < 50.0 OR (TOD_TO_UDINT(UDINT_TO_TOD(VI_System_Time_MS)) > 64800000 OR TOD_TO_UDINT(UDINT_TO_TOD(VI_System_Time_MS)) < 28800000)) THEN
    IF VI_Motion_Corridor OR (L_State = 2) THEN VO_Light_Corridor := TRUE; VO_Light_Stairs_Dim := 30;
    ELSE VO_Light_Corridor := FALSE; VO_Light_Stairs_Dim := 0; END_IF;
END_IF;

END_FUNCTION_BLOCK

// POUs/FB_Water_Leakage_Manager
FUNCTION_BLOCK FB_Water_Leakage_Manager
VAR_INPUT
    VI_System_Time_MS : UDINT;
    VI_IsActivePLC : BOOL;
    VI_Sensors : ARRAY[1..12] OF BOOL;
    VI_Valve_35_Current : REAL;
    VI_Valve_36_Current : REAL;
    VI_Emergency_Open_Req : BYTE; // 1, 3, 5 мин
    VI_Config : ST_Flood_Config; // ТЗ 4.4
    VI_Power_OK : BOOL; // ТЗ 4.3: Мониторинг питания
    VI_Two_Stage_Confirm : BOOL; // ТЗ 4.4: Подтверждение
END_VAR
VAR_OUTPUT
    VO_Valve_35_Close : BOOL;
    VO_Valve_36_Close : BOOL;
    VO_Flood_Alarm : BOOL;
    VO_Alert_Priority : BYTE; // ТЗ 4.3: 1-Low, 2-Normal, 3-Critical
    VO_Status_Msg : STRING(200);
END_VAR
VAR
    L_Zone1_Alarm : BOOL;
    L_Zone2_Alarm : BOOL;
    L_Zone3_Alarm : BOOL;
    L_Emergency_Timer : TON;
    L_Confirm_Timer : TON;
    L_Confirm_Wait : BOOL;
    
    // ТЗ 4.4: Лимит 3 раза в сутки
    L_Emergency_Count : UINT;
    L_Day_Timer : TON;
    L_Last_Req : BYTE;
    
    // ТЗ 4.3: Диагностика тока
    L_Valve_35_Error : BOOL;
    L_Valve_36_Error : BOOL;
END_VAR

// 1. Определение протечки по зонам (ТЗ 4.1)
L_Zone1_Alarm := VI_Sensors[1] OR VI_Sensors[2] OR VI_Sensors[3];
L_Zone2_Alarm := VI_Sensors[4] OR VI_Sensors[5];
L_Zone3_Alarm := VI_Sensors[6] OR VI_Sensors[7];
VO_Flood_Alarm := L_Zone1_Alarm OR L_Zone2_Alarm OR L_Zone3_Alarm;

// 2. Управление клапанами (ТЗ 4.2, 4.3)
// ТЗ 4.3: НЗ клапаны закрываются при потере питания (автоматически физически)
// Но мы должны отразить это в логике и статусе
VO_Valve_35_Close := L_Zone1_Alarm OR NOT VI_Power_OK;
VO_Valve_36_Close := L_Zone2_Alarm OR L_Zone3_Alarm OR NOT VI_Power_OK;

// Диагностика по току (ТЗ 4.3)
L_Valve_35_Error := (VO_Valve_35_Close AND VI_Valve_35_Current < 50.0) OR (NOT VO_Valve_35_Close AND VI_Valve_35_Current > VI_Config.Current_Threshold_MA);
L_Valve_36_Error := (VO_Valve_36_Close AND VI_Valve_36_Current < 50.0) OR (NOT VO_Valve_36_Close AND VI_Valve_36_Current > VI_Config.Current_Threshold_MA);

// Эскалация приоритета (ТЗ 4.3)
IF VO_Flood_Alarm THEN
    VO_Alert_Priority := 2; // Normal
    IF L_Valve_35_Error OR L_Valve_36_Error THEN
        VO_Alert_Priority := 3; // Critical (НО клапан не закрылся или обрыв)
    END_IF;
ELSE
    VO_Alert_Priority := 1; // Low
END_IF;

// 3. Экстренное открытие (ТЗ 4.4)
L_Day_Timer(IN := TRUE, PT := T#24h);
IF L_Day_Timer.Q THEN L_Emergency_Count := 0; L_Day_Timer(IN := FALSE); END_IF;

IF VI_Emergency_Open_Req > 0 AND VI_Emergency_Open_Req <> L_Last_Req AND L_Emergency_Count < 3 THEN
    IF VI_Config.Emergency_Two_Stage_Enabled AND NOT L_Confirm_Wait THEN
        L_Confirm_Wait := TRUE;
        L_Confirm_Timer(IN := TRUE, PT := T#30s);
        VO_Status_Msg := 'ОЖИДАНИЕ ПОДТВЕРЖДЕНИЯ ЭКСТРЕННОГО ОТКРЫТИЯ';
    ELSIF (VI_Config.Emergency_Two_Stage_Enabled AND VI_Two_Stage_Confirm) OR NOT VI_Config.Emergency_Two_Stage_Enabled THEN
        L_Emergency_Count := L_Emergency_Count + 1;
        L_Last_Req := VI_Emergency_Open_Req;
        L_Emergency_Timer(IN := TRUE, PT := TO_TIME(TO_UDINT(VI_Emergency_Open_Req) * 60000));
        L_Confirm_Wait := FALSE; L_Confirm_Timer(IN := FALSE);
    END_IF;
END_IF;

L_Confirm_Timer(IN := L_Confirm_Wait);
IF L_Confirm_Timer.Q THEN L_Confirm_Wait := FALSE; L_Confirm_Timer(IN := FALSE); END_IF;

IF L_Emergency_Timer.IN AND NOT L_Emergency_Timer.Q THEN
    VO_Valve_35_Close := FALSE; VO_Valve_36_Close := FALSE;
    VO_Status_Msg := 'ЭКСТРЕННОЕ ОТКРЫТИЕ ВОДЫ';
ELSE
    L_Emergency_Timer(IN := FALSE);
    IF VI_Emergency_Open_Req = 0 THEN L_Last_Req := 0; END_IF;
END_IF;

IF VO_Flood_Alarm AND NOT L_Emergency_Timer.IN AND NOT L_Confirm_Wait THEN VO_Status_Msg := 'ОБНАРУЖЕНА ПРОТЕЧКА ВОДЫ'; END_IF;
IF NOT VI_Power_OK THEN VO_Status_Msg := 'ВНИМАНИЕ: ОТСУТСТВИЕ ПИТАНИЯ КЛАПАНОВ'; END_IF;

END_FUNCTION_BLOCK

// POUs/FB_Gas_Smoke_Manager
FUNCTION_BLOCK FB_Gas_Smoke_Manager
VAR_INPUT
    VI_System_Time_MS : UDINT;
    VI_IsActivePLC : BOOL;
    VI_Methane_LEL : ARRAY[1..2] OF REAL;
    VI_CO_PPM : ARRAY[1..8] OF REAL;
    VI_Smoke_Sensors : ARRAY[1..6] OF BOOL;
    VI_Mute_Request : BOOL;
END_VAR
VAR_OUTPUT
    VO_Gas_Alarm : BOOL;
    VO_Fire_Alarm : BOOL;
    VO_Siren_Active : BOOL;
    VO_Gas_Valve_Close : BOOL;
    VO_Boiler_Stop : BOOL;
    VO_Vent_PV3_Boost : BOOL; // ТЗ 5.1 (ПВ-3 при 10% LEL)
    VO_Supply_100_Req : BOOL; // ТЗ 6.4 (Метан >20%)
    VO_Exhaust_100_Req : BOOL; // ТЗ 6.4 (Пожар)
    VO_Supply_80_Req : BOOL; // ТЗ 5.4 (CO)
    VO_Status_Msg : STRING(200);
END_VAR
VAR
    L_Methane_Max : REAL;
    L_CO_Max : REAL;
    L_Smoke_Active : BOOL;
    L_Smoke_Timer : ARRAY[1..6] OF TON;
    L_Mute_Timer : TON;
    L_Muted : BOOL;
    L_Mute_Count : UINT; // ТЗ 5.5
    L_i : INT;
    L_j : INT;
    L_Smoke_Count : UINT;
    
    // ТЗ 5.2: Временные пороги CO
    L_CO_Timer_30ppm : TON; // 8 часов
    L_CO_Timer_70ppm : TON; // 1 час
    L_CO_Timer_400ppm : TON; // 15 минут
END_VAR

// 1. Обработка метана (ТЗ 5.1, 6.4)
L_Methane_Max := 0.0;
FOR L_i := 1 TO 2 DO IF VI_Methane_LEL[L_i] > L_Methane_Max THEN L_Methane_Max := VI_Methane_LEL[L_i]; END_IF; END_FOR;

VO_Vent_PV3_Boost := (L_Methane_Max >= 10.0); // ТЗ 5.1: ПВ-3 при 10% LEL

IF L_Methane_Max >= 40.0 THEN
    VO_Gas_Alarm := TRUE; VO_Gas_Valve_Close := TRUE; VO_Boiler_Stop := TRUE; VO_Supply_100_Req := TRUE;
    VO_Status_Msg := 'КРИТИЧЕСКАЯ УТЕЧКА ГАЗА (40% LEL)';
ELSIF L_Methane_Max >= 20.0 THEN
    VO_Gas_Alarm := TRUE; VO_Gas_Valve_Close := TRUE; VO_Boiler_Stop := TRUE; VO_Supply_100_Req := TRUE;
    VO_Status_Msg := 'УТЕЧКА ГАЗА (20% LEL)';
ELSIF L_Methane_Max >= 10.0 THEN 
    VO_Status_Msg := 'ПРЕДУПРЕЖДЕНИЕ: ГАЗ (10% LEL)';
END_IF;

// 2. Обработка CO (ТЗ 5.2, 5.4)
L_CO_Max := 0.0;
FOR L_i := 1 TO 8 DO IF VI_CO_PPM[L_i] > L_CO_Max THEN L_CO_Max := VI_CO_PPM[L_i]; END_IF; END_FOR;

L_CO_Timer_30ppm(IN := (L_CO_Max >= 30.0), PT := T#8h);
L_CO_Timer_70ppm(IN := (L_CO_Max >= 70.0), PT := T#1h);
L_CO_Timer_400ppm(IN := (L_CO_Max >= 400.0), PT := T#15m);

IF L_CO_Timer_400ppm.Q THEN VO_Gas_Alarm := TRUE; VO_Status_Msg := 'КРИТИЧЕСКАЯ КОНЦЕНТРАЦИЯ CO (400 ppm / 15 мин)';
ELSIF L_CO_Timer_70ppm.Q THEN VO_Gas_Alarm := TRUE; VO_Status_Msg := 'ВЫСОКАЯ КОНЦЕНТРАЦИЯ CO (70 ppm / 1 час)';
ELSIF L_CO_Timer_30ppm.Q THEN VO_Gas_Alarm := TRUE; VO_Status_Msg := 'ПОВЫШЕННАЯ КОНЦЕНТРАЦИЯ CO (30 ppm / 8 час)';
END_IF;

IF VO_Gas_Alarm AND L_CO_Max >= 30.0 THEN VO_Supply_80_Req := TRUE; END_IF; // ТЗ 5.4

// 3. Обработка дыма (ТЗ 5.3, 6.4)
L_Smoke_Count := 0;
FOR L_i := 1 TO 6 DO
    L_Smoke_Timer[L_i](IN := VI_Smoke_Sensors[L_i], PT := T#30s);
    IF VI_Smoke_Sensors[L_i] THEN L_Smoke_Count := L_Smoke_Count + 1; END_IF;
    // ТЗ 5.3: Верификация вторым датчиком ИЛИ сигнал > 30 сек
    IF L_Smoke_Timer[L_i].Q OR (L_Smoke_Count >= 2) THEN L_Smoke_Active := TRUE; END_IF;
END_FOR;

IF L_Smoke_Active THEN 
    VO_Fire_Alarm := TRUE; VO_Boiler_Stop := TRUE; VO_Exhaust_100_Req := TRUE;
    VO_Status_Msg := 'ПОЖАРНАЯ ТРЕВОГА: ДЫМ'; 
END_IF;

// 4. Сирена и квитирование (ТЗ 5.5)
IF VO_Gas_Alarm OR VO_Fire_Alarm THEN
    IF VI_Mute_Request AND NOT L_Muted AND L_Mute_Count < 3 THEN
        L_Muted := TRUE; L_Mute_Count := L_Mute_Count + 1;
        L_Mute_Timer(IN := TRUE, PT := T#5m);
    END_IF;
    
    L_Mute_Timer(IN := L_Muted);
    IF L_Mute_Timer.Q THEN L_Muted := FALSE; L_Mute_Timer(IN := FALSE); END_IF;
    VO_Siren_Active := NOT L_Muted;
ELSE
    L_Muted := FALSE; L_Mute_Count := 0; VO_Siren_Active := FALSE;
END_IF;

END_FUNCTION_BLOCK

// POUs/FB_Ventilation_System_Manager
FUNCTION_BLOCK FB_Ventilation_System_Manager
VAR_INPUT
    VI_System_Time_MS : UDINT;
    VI_IsActivePLC : BOOL;
    VI_CO2 : ARRAY[1..8] OF REAL;
    VI_Humidity : ARRAY[1..8] OF REAL;
    VI_Gas_Alarm : BOOL;
    VI_Fire_Alarm : BOOL;
    VI_Flood_Alarm : BOOL;
    VI_Config : ST_Ventilation_Config;
    VI_PV3_Boost : BOOL; // ТЗ 5.1
    VI_Supply_100_Req : BOOL; // ТЗ 6.4
    VI_Exhaust_100_Req : BOOL; // ТЗ 6.4
    VI_Supply_80_Req : BOOL; // ТЗ 5.4
    VI_Wet_Zone_Lights : ARRAY[1..4] OF BOOL; // ТЗ 4.0
END_VAR
VAR_OUTPUT
    VO_Supply_Fans : ARRAY[1..3] OF REAL; // 0-100%
    VO_Exhaust_Fans : ARRAY[1..5] OF REAL; // 0-100%
    VO_Status : ARRAY[1..8] OF ST_Ventilation_Unit;
END_VAR
VAR
    L_Mode : BYTE; // 0-Eco, 1-Std, 2-Int, 3-Emergency
    L_Base_Speed : REAL;
    L_i : INT;
    L_Max_CO2 : REAL;
    L_Max_Hum : REAL;
    L_Is_Night : BOOL;
    L_Current_Time : TOD;
    L_Wet_Zone_Timers : ARRAY[1..4] OF TON;
END_VAR

// 1. Определение режима
L_Current_Time := UDINT_TO_TOD(VI_System_Time_MS MOD 86400000);
L_Is_Night := (L_Current_Time >= VI_Config.Night_Mode_Start OR L_Current_Time <= VI_Config.Night_Mode_End);

// Поиск максимумов
L_Max_CO2 := 0.0;
FOR L_i := 1 TO 8 DO
    IF VI_CO2[L_i] > L_Max_CO2 THEN L_Max_CO2 := VI_CO2[L_i]; END_IF;
END_FOR;

L_Max_Hum := 0.0;
FOR L_i := 1 TO 8 DO
    IF VI_Humidity[L_i] > L_Max_Hum THEN L_Max_Hum := VI_Humidity[L_i]; END_IF;
END_FOR;

// Выбор режима (ТЗ 6.3)
IF VI_Gas_Alarm OR VI_Fire_Alarm OR VI_Flood_Alarm THEN
    L_Mode := 3; // Аварийный
    L_Base_Speed := 100.0;
ELSIF L_Max_CO2 > VI_Config.CO2_Threshold OR L_Max_Hum > VI_Config.Humidity_Threshold THEN
    L_Mode := 2; // Интенсив
    L_Base_Speed := 70.0;
ELSIF L_Is_Night THEN
    L_Mode := 0; // Эконом
    L_Base_Speed := 20.0;
ELSE
    L_Mode := 1; // Стандарт
    L_Base_Speed := 40.0;
END_IF;

// 2. Управление вентиляторами
FOR L_i := 1 TO 3 DO
    VO_Supply_Fans[L_i] := L_Base_Speed;
    
    // ТЗ 5.4: CO -> приток 80%
    IF VI_Supply_80_Req THEN VO_Supply_Fans[L_i] := 80.0; END_IF;
    
    // ТЗ 6.4: Метан >20% -> приток 100%
    IF VI_Supply_100_Req THEN VO_Supply_Fans[L_i] := 100.0; END_IF;

    // ТЗ 5.1: ПВ-3 форсирован при 10% LEL
    IF L_i = 3 AND VI_PV3_Boost THEN VO_Supply_Fans[L_i] := 100.0; END_IF;

    // Интеграция с безопасностью (ТЗ 6.4): При пожаре приток ОТКЛЮЧАЕТСЯ
    IF VI_Fire_Alarm THEN
        VO_Supply_Fans[L_i] := 0.0;
    END_IF;
END_FOR;

FOR L_i := 1 TO 5 DO
    VO_Exhaust_Fans[L_i] := L_Base_Speed;
    
    // ТЗ 4.0: Интеграция с мокрыми зонами (вытяжки 4-5)
    IF L_i >= 4 THEN
        L_Wet_Zone_Timers[L_i-3](IN := VI_Wet_Zone_Lights[L_i-3], PT := T#7m); // 7 мин пост-вентиляция
        IF L_Wet_Zone_Timers[L_i-3].Q THEN
            VO_Exhaust_Fans[L_i] := MAX(VO_Exhaust_Fans[L_i], 60.0); // Форсируем вытяжку
        END_IF;
    END_IF;

    // ТЗ 6.4: Пожар -> вытяжка 100%
    IF VI_Exhaust_100_Req THEN VO_Exhaust_Fans[L_i] := 100.0; END_IF;
END_FOR;

// 3. Статус
FOR L_i := 1 TO 3 DO
    VO_Status[L_i].Enabled := VI_IsActivePLC;
    VO_Status[L_i].Speed_Percent := VO_Supply_Fans[L_i];
    VO_Status[L_i].Mode := L_Mode;
END_FOR;

END_FUNCTION_BLOCK

// POUs/FB_User_Rule_Engine
FUNCTION_BLOCK FB_User_Rule_Engine
VAR_INPUT
    VI_Rules : ARRAY[1..10] OF ST_User_Rule;
    VI_System_State : ST_System_State_Summary; // Текущие значения всех датчиков
END_VAR
VAR_OUTPUT
    VO_Actions : ARRAY[1..10] OF ST_Rule_Action;
END_VAR
VAR
    L_i : INT;
    L_Condition_Met : BOOL;
    L_Val : REAL;
    L_Applied_Priority : ARRAY[1..100] OF BYTE; // Приоритет примененного действия для Target_ID
END_VAR

// Сброс приоритетов перед циклом
FOR L_i := 1 TO 100 DO L_Applied_Priority[L_i] := 0; END_FOR;

FOR L_i := 1 TO 10 DO
    IF VI_Rules[L_i].Enabled THEN
        L_Condition_Met := FALSE;
        
        // Вычисление условия (ТЗ 7.4)
        CASE VI_Rules[L_i].Condition_Type OF
            1: // Температура уличная
                L_Val := VI_System_State.Outdoor_Temp;
            2: // Температура пола (Зона 1)
                L_Val := VI_System_State.Floor_Temps[1];
            3: // CO2 (Зона 1)
                L_Val := VI_System_State.CO2[1];
            4: // Охрана
                L_Val := SEL(VI_System_State.Security_Armed, 0.0, 1.0);
        END_CASE;

        CASE VI_Rules[L_i].Condition_Op OF
            1: L_Condition_Met := (L_Val > VI_Rules[L_i].Condition_Value);
            2: L_Condition_Met := (L_Val < VI_Rules[L_i].Condition_Value);
            3: L_Condition_Met := (ABS(L_Val - VI_Rules[L_i].Condition_Value) < 0.01);
        END_CASE;

        // Выполнение действия с учетом приоритета (ТЗ 7.4)
        IF L_Condition_Met THEN
             // Проверяем, не выполнялось ли уже действие для этого Target_ID с более высоким приоритетом
             IF VI_Rules[L_i].Action_Target_ID > 0 AND VI_Rules[L_i].Action_Target_ID <= 100 THEN
                 IF VI_Rules[L_i].Priority >= L_Applied_Priority[VI_Rules[L_i].Action_Target_ID] THEN
                     VO_Actions[L_i].Active := TRUE;
                     VO_Actions[L_i].Target_ID := VI_Rules[L_i].Action_Target_ID;
                     VO_Actions[L_i].Value := VI_Rules[L_i].Action_Value;
                     L_Applied_Priority[VI_Rules[L_i].Action_Target_ID] := VI_Rules[L_i].Priority;
                 ELSE
                     VO_Actions[L_i].Active := FALSE; // Игнорируем из-за низкого приоритета
                 END_IF;
             END_IF;
        ELSE
             VO_Actions[L_i].Active := FALSE;
        END_IF;
    END_IF;
END_FOR;

END_FUNCTION_BLOCK

// POUs/FB_Lighting_Blinds_Manager
FUNCTION_BLOCK FB_Lighting_Blinds_Manager
VAR_INPUT
    VI_System_Time_MS : UDINT;
    VI_IsActivePLC : BOOL;
    VI_Current_Scenario : E_SCENARIO_TYPE;
    VI_Away_Level : BYTE; // 1-Short, 2-Medium, 3-Long
    VI_Simulation_Active : BOOL;
    VI_Manual_Light_Override : ARRAY[1..16] OF BYTE; // 0-100
    VI_Manual_Blinds_Override : ARRAY[1..20] OF BYTE; // 0-100
    VI_Simulation_Lights : ARRAY[1..16] OF BOOL;
    VI_Physical_Switches : ARRAY[1..16] OF BOOL; // ТЗ 1.0
    VI_Motion_Sensors : ARRAY[1..16] OF BOOL; // ТЗ 2.0
    VI_Maintenance : ARRAY[1..16] OF ST_Component_Maintenance; // ТЗ 6.0
END_VAR
VAR_OUTPUT
    VO_Lighting_Levels : ARRAY[1..16] OF BYTE;
    VO_Blinds_Positions : ARRAY[1..20] OF BYTE;
    VO_Wet_Zone_Light_Active : ARRAY[1..4] OF BOOL; // Для вентиляции (ТЗ 4.0)
END_VAR
VAR
    L_i : INT;
    L_Base_Light : BYTE;
    L_Base_Blinds : BYTE;
    L_Light_States : ARRAY[1..16] OF BOOL;
    L_Prev_Switches : ARRAY[1..16] OF BOOL;
    L_Motion_Timers : ARRAY[1..16] OF TON;
END_VAR

// 1. Определение базовых уровней по сценарию (ТЗ 7.1)
CASE VI_Current_Scenario OF
    E_SCENARIO_TYPE.SCENARIO_MORNING:
        L_Base_Light := 70;
        L_Base_Blinds := 80; // 80% открыты
    
    E_SCENARIO_TYPE.SCENARIO_EVENING:
        L_Base_Light := 40;
        L_Base_Blinds := 10; // 90% закрыты (10% открыты)
        
    E_SCENARIO_TYPE.SCENARIO_AWAY:
        L_Base_Light := 0;
        L_Base_Blinds := 0; // 100% закрыты
        
    ELSE
        L_Base_Light := 100;
        L_Base_Blinds := 100;
END_CASE;

// 2. Управление освещением
FOR L_i := 1 TO 16 DO
    // Приоритет 1: Физические выключатели (ТЗ 1.0)
    IF VI_Physical_Switches[L_i] AND NOT L_Prev_Switches[L_i] THEN
        L_Light_States[L_i] := NOT L_Light_States[L_i];
    END_IF;
    L_Prev_Switches[L_i] := VI_Physical_Switches[L_i];

    // Приоритет 2: Датчики движения (ТЗ 2.0)
    L_Motion_Timers[L_i](IN := VI_Motion_Sensors[L_i], PT := T#5m);
    IF VI_Motion_Sensors[L_i] THEN
        L_Light_States[L_i] := TRUE;
    ELSIF L_Motion_Timers[L_i].Q THEN
        L_Light_States[L_i] := FALSE;
    END_IF;

    // Приоритет 3: Симуляция (только в режиме Away)
    IF VI_Current_Scenario = E_SCENARIO_TYPE.SCENARIO_AWAY AND VI_Simulation_Active THEN
        L_Light_States[L_i] := VI_Simulation_Lights[L_i];
    END_IF;

    // Приоритет 4: Ремонт/Неисправность (ТЗ 6.0, 7.0)
    IF VI_Maintenance[L_i].Is_Faulty OR VI_Maintenance[L_i].Is_In_Maintenance THEN
        VO_Lighting_Levels[L_i] := REAL_TO_BYTE(VI_Maintenance[L_i].Fallback_Value);
    ELSE
        VO_Lighting_Levels[L_i] := SEL(L_Light_States[L_i], 0, L_Base_Light);
    END_IF;
    
    // 5. Мокрые зоны (допустим зоны 13-16 - санузлы)
    IF L_i >= 13 THEN
        VO_Wet_Zone_Light_Active[L_i - 12] := (VO_Lighting_Levels[L_i] > 10);
    END_IF;
END_FOR;

// 3. Управление шторами
FOR L_i := 1 TO 20 DO
    // Приоритет 1: Ручное управление
    IF VI_Manual_Blinds_Override[L_i] > 0 THEN
        VO_Blinds_Positions[L_i] := VI_Manual_Blinds_Override[L_i];
    // Приоритет 2: Сценарий
    ELSE
        VO_Blinds_Positions[L_i] := L_Base_Blinds;
    END_IF;
END_FOR;

END_FUNCTION_BLOCK

// POUs/FB_Simulation_Manager
FUNCTION_BLOCK FB_Simulation_Manager
VAR_INPUT
    VI_System_Time_MS : UDINT;
    VI_Enabled : BOOL;
    VI_Intensity : REAL; // 0.2-0.3
END_VAR
VAR_OUTPUT
    VO_Light_States : ARRAY[1..16] OF BOOL;
    VO_Socket_States : ARRAY[1..12] OF BOOL;
END_VAR
VAR
    L_Rand : FB_Random_Generator;
    L_Last_Event_Time : UDINT;
    L_Event_Duration : UDINT;
    L_Active : BOOL;
    L_i : INT;
    L_Current_TOD : TOD;
    L_In_Window : BOOL;
END_VAR

IF NOT VI_Enabled THEN L_Active := FALSE; RETURN; END_IF;

// ТЗ 7.2: Временные окна (07-10, 18-23, 01-04)
L_Current_TOD := UDINT_TO_TOD(VI_System_Time_MS MOD 86400000);
L_In_Window := (L_Current_TOD >= TOD#07:00 AND L_Current_TOD <= TOD#10:00) OR
               (L_Current_TOD >= TOD#18:00 AND L_Current_TOD <= TOD#23:00) OR
               (L_Current_TOD >= TOD#01:00 AND L_Current_TOD <= TOD#04:00);

IF NOT L_In_Window THEN L_Active := FALSE; FOR L_i := 1 TO 16 DO VO_Light_States[L_i] := FALSE; END_FOR; RETURN; END_IF;

// Логика случайных событий
IF NOT L_Active THEN
    IF (L_Rand.Random_Int_Range(0, 1000) < TO_UDINT(VI_Intensity * 10.0)) THEN
        L_Active := TRUE; L_Last_Event_Time := VI_System_Time_MS;
        
        // ТЗ 7.2: Распределение 70/30
        IF L_Rand.Random_Int_Range(0, 100) < 70 THEN
            L_Event_Duration := L_Rand.Random_Int_Range(300000, 900000); // 5-15 мин (70%)
        ELSE
            L_Event_Duration := L_Rand.Random_Int_Range(900001, 2700000); // 15-45 мин (30%)
        END_IF;
        
        FOR L_i := 1 TO 16 DO VO_Light_States[L_i] := (L_Rand.Random_Int_Range(0, 10) > 7); END_FOR;
    END_IF;
ELSE
    IF (VI_System_Time_MS - L_Last_Event_Time) >= L_Event_Duration THEN
        L_Active := FALSE; FOR L_i := 1 TO 16 DO VO_Light_States[L_i] := FALSE; END_FOR;
    END_IF;
END_IF;

END_FUNCTION_BLOCK

// POUs/FB_Random_Generator
FUNCTION_BLOCK FB_Random_Generator
VAR
    L_seed : UDINT := 1;
END_VAR
VAR CONSTANT
    C_LCG_MULTIPLIER : UDINT := 1664525;
    C_LCG_INCREMENT  : UDINT := 1013904223;
    C_LCG_MODULUS    : LREAL := 4294967296.0;
END_VAR

METHOD Random_Int_Range : UDINT
VAR_INPUT
    VI_min : UDINT;
    VI_max : UDINT;
END_VAR
VAR
    L_range : UDINT;
    L_rand_factor : LREAL;
END_VAR
L_seed := (C_LCG_MULTIPLIER * L_seed) + C_LCG_INCREMENT;

IF VI_max > VI_min THEN
        L_range := VI_max - VI_min;
        // Используем LREAL для точности и исключения выхода за границу
        L_rand_factor := TO_LREAL(L_seed) / C_LCG_MODULUS;
        Random_Int_Range := VI_min + TO_UDINT(L_rand_factor * TO_LREAL(L_range + 1));
        
        // Финальная защита от переполнения
        IF Random_Int_Range > VI_max THEN
            Random_Int_Range := VI_max;
        END_IF;
    ELSE
        Random_Int_Range := VI_min;
    END_IF;
END_METHOD

END_FUNCTION_BLOCK

// POUs/FB_DHW_Manager
FUNCTION_BLOCK FB_DHW_Manager
VAR_INPUT
    VI_System_Time_MS : UDINT;
    VI_IsActivePLC : BOOL;
    VI_Temp : REAL;
    VI_Pressure : REAL;
    VI_Config : ST_DHW_Config;
    VI_Maintenance : ST_Component_Maintenance;
END_VAR
VAR_OUTPUT
    VO_Status : ST_DHW_Status;
    VO_Heating_Pump : BOOL;
    VO_Circ_Pump : BOOL;
END_VAR
VAR
    L_Current_TOD : TOD;
    L_Legionella_Active : BOOL;
    L_Last_Good_Temp : REAL := 55.0;
END_VAR

// 1. Обработка неисправности (ТЗ 7.0)
IF VI_Maintenance.Is_Faulty OR VI_Maintenance.Is_In_Maintenance THEN
    VO_Status.Temp := SEL(VI_Maintenance.Use_Last_Good_Value, VI_Maintenance.Fallback_Value, L_Last_Good_Temp);
ELSE
    VO_Status.Temp := VI_Temp;
    L_Last_Good_Temp := VI_Temp;
END_IF;

VO_Status.Pressure := VI_Pressure;

// 2. Логика нагрева
IF VI_IsActivePLC THEN
    IF VO_Status.Temp < (VI_Config.Target_Temp - VI_Config.Hysteresis) THEN
        VO_Heating_Pump := TRUE;
    ELSIF VO_Status.Temp > (VI_Config.Target_Temp + VI_Config.Hysteresis) THEN
        VO_Heating_Pump := FALSE;
    END_IF;
    
    // 3. Циркуляция ГВС по расписанию
    L_Current_TOD := UDINT_TO_TOD(VI_System_Time_MS MOD 86400000);
    VO_Circ_Pump := VI_Config.Circulation_Schedule_Enabled AND 
                    (L_Current_TOD >= VI_Config.Circulation_Start AND L_Current_TOD <= VI_Config.Circulation_End);
ELSE
    VO_Heating_Pump := FALSE;
    VO_Circ_Pump := FALSE;
END_IF;

VO_Status.Heating_Pump_On := VO_Heating_Pump;
VO_Status.Circ_Pump_On := VO_Circ_Pump;
VO_Status.Error := (VI_Pressure < 1.0 OR VI_Pressure > 4.0);

END_FUNCTION_BLOCK

// POUs/FB_Access_Control
FUNCTION_BLOCK FB_Access_Control
VAR_INPUT
    VI_System_Time_MS   : UDINT;
    VI_IsActivePLC      : BOOL;
    VI_Armed            : BOOL; // Состояние охраны
    
    // Команды HMI
    VI_Gate_Open_Req    : BOOL;
    VI_Wicket_Open_Req  : BOOL;
    VI_Lock_1_Open_Req  : BOOL;
    VI_Lock_1_Close_Req : BOOL;
    VI_Lock_2_Open_Req  : BOOL;
    VI_Lock_2_Close_Req : BOOL;
    
    // Настройки
    VI_Config           : ST_Security_Config;
END_VAR
VAR_OUTPUT
    VO_Gate_Open        : BOOL;
    VO_Wicket_Open      : BOOL;
    VO_Lock_1_Open      : BOOL;
    VO_Lock_1_Close     : BOOL;
    VO_Lock_2_Open      : BOOL;
    VO_Lock_2_Close     : BOOL;
END_VAR
VAR
    L_Gate_Timer        : TON;
    L_Wicket_Timer      : TON;
    L_Lock_1_Open_T     : TON;
    L_Lock_1_Close_T    : TON;
    L_Lock_2_Open_T     : TON;
    L_Lock_2_Close_T    : TON;
    
    L_Prev_Armed        : BOOL;
    L_Auto_Lock_Req     : BOOL;
END_VAR

IF NOT VI_IsActivePLC THEN
    RETURN;
END_IF;

// 1. Автоматическое закрытие при постановке на охрану
IF VI_Armed AND NOT L_Prev_Armed THEN
    L_Auto_Lock_Req := TRUE;
END_IF;
L_Prev_Armed := VI_Armed;

// 2. Логика импульсов
// Ворота
L_Gate_Timer(IN := VI_Gate_Open_Req, PT := TO_TIME(VI_Config.gate_open_pulse_ms));
VO_Gate_Open := VI_Gate_Open_Req AND NOT L_Gate_Timer.Q;

// Калитка
L_Wicket_Timer(IN := VI_Wicket_Open_Req, PT := TO_TIME(VI_Config.wicket_open_pulse_ms));
VO_Wicket_Open := VI_Wicket_Open_Req AND NOT L_Wicket_Timer.Q;

// Замок 1
L_Lock_1_Open_T(IN := VI_Lock_1_Open_Req, PT := TO_TIME(VI_Config.lock_open_pulse_ms));
VO_Lock_1_Open := VI_Lock_1_Open_Req AND NOT L_Lock_1_Open_T.Q;

L_Lock_1_Close_T(IN := (VI_Lock_1_Close_Req OR L_Auto_Lock_Req), PT := TO_TIME(VI_Config.lock_close_pulse_ms));
VO_Lock_1_Close := (VI_Lock_1_Close_Req OR L_Auto_Lock_Req) AND NOT L_Lock_1_Close_T.Q;

// Замок 2
L_Lock_2_Open_T(IN := VI_Lock_2_Open_Req, PT := TO_TIME(VI_Config.lock_open_pulse_ms));
VO_Lock_2_Open := VI_Lock_2_Open_Req AND NOT L_Lock_2_Open_T.Q;

L_Lock_2_Close_T(IN := (VI_Lock_2_Close_Req OR L_Auto_Lock_Req), PT := TO_TIME(VI_Config.lock_close_pulse_ms));
VO_Lock_2_Close := (VI_Lock_2_Close_Req OR L_Auto_Lock_Req) AND NOT L_Lock_2_Close_T.Q;

// Сброс авто-закрытия после завершения импульса
IF L_Lock_1_Close_T.Q AND L_Lock_2_Close_T.Q THEN
    L_Auto_Lock_Req := FALSE;
END_IF;

END_FUNCTION_BLOCK

// POUs/FB_PLC_Heartbeat
FUNCTION_BLOCK FB_PLC_Heartbeat
VAR_INPUT
    VI_Local_ID : BYTE;
    VI_System_Time : UDINT;
    VI_Remote_Pulse : BOOL;
    VI_Remote_Is_Active : BOOL; // ТЗ 8.3: Уровень 2 - проверка роли партнера
    VI_Gateway_Ping_OK : BOOL; // ТЗ 8.3: Уровень 3 - пинг шлюза
END_VAR
VAR_OUTPUT
    VO_Is_Active : BOOL;
    VO_RTT_MS : UDINT;
    VO_Loss_Count : UDINT; // ТЗ 8.4: Статистика потерь
    VO_Max_RTT : UDINT; // ТЗ 8.4: Макс. задержка
END_VAR
VAR
    L_Last_Pulse : BOOL;
    L_Last_Pulse_Time : UDINT;
    L_Timeout : UDINT := 500; // ТЗ 8.1: 500 мс
    L_Pulse_Send_Time : UDINT;
    L_Loss_Timer : TON;
END_VAR

// 1. Мониторинг пульса и RTT (ТЗ 8.4)
IF VI_Remote_Pulse <> L_Last_Pulse THEN
    VO_RTT_MS := VI_System_Time - L_Last_Pulse_Time;
    IF VO_RTT_MS > VO_Max_RTT THEN VO_Max_RTT := VO_RTT_MS; END_IF;
    L_Last_Pulse := VI_Remote_Pulse;
    L_Last_Pulse_Time := VI_System_Time;
END_IF;

L_Loss_Timer(IN := (VI_System_Time - L_Last_Pulse_Time) > L_Timeout, PT := T#1s);
IF L_Loss_Timer.Q THEN 
    VO_Loss_Count := VO_Loss_Count + 1; 
    L_Loss_Timer(IN := FALSE); 
END_IF;

// 2. Логика активности и защита от раскола мозга (ТЗ 8.3)
// Уровень 1: Тайм-аут пульса
IF (VI_System_Time - L_Last_Pulse_Time) < L_Timeout THEN
    // Уровень 2: Если партнер заявляет, что он активен, и у него приоритет (ID=1)
    IF VI_Remote_Is_Active AND VI_Local_ID = 2 THEN
        VO_Is_Active := FALSE;
    ELSE
        // Приоритет у ПЛК A (ID=1)
        VO_Is_Active := (VI_Local_ID = 1);
    END_IF;
ELSE
    // Уровень 3: Если связи нет, проверяем доступность шлюза
    VO_Is_Active := VI_Gateway_Ping_OK OR (VI_Local_ID = 1);
END_IF;

END_FUNCTION_BLOCK

